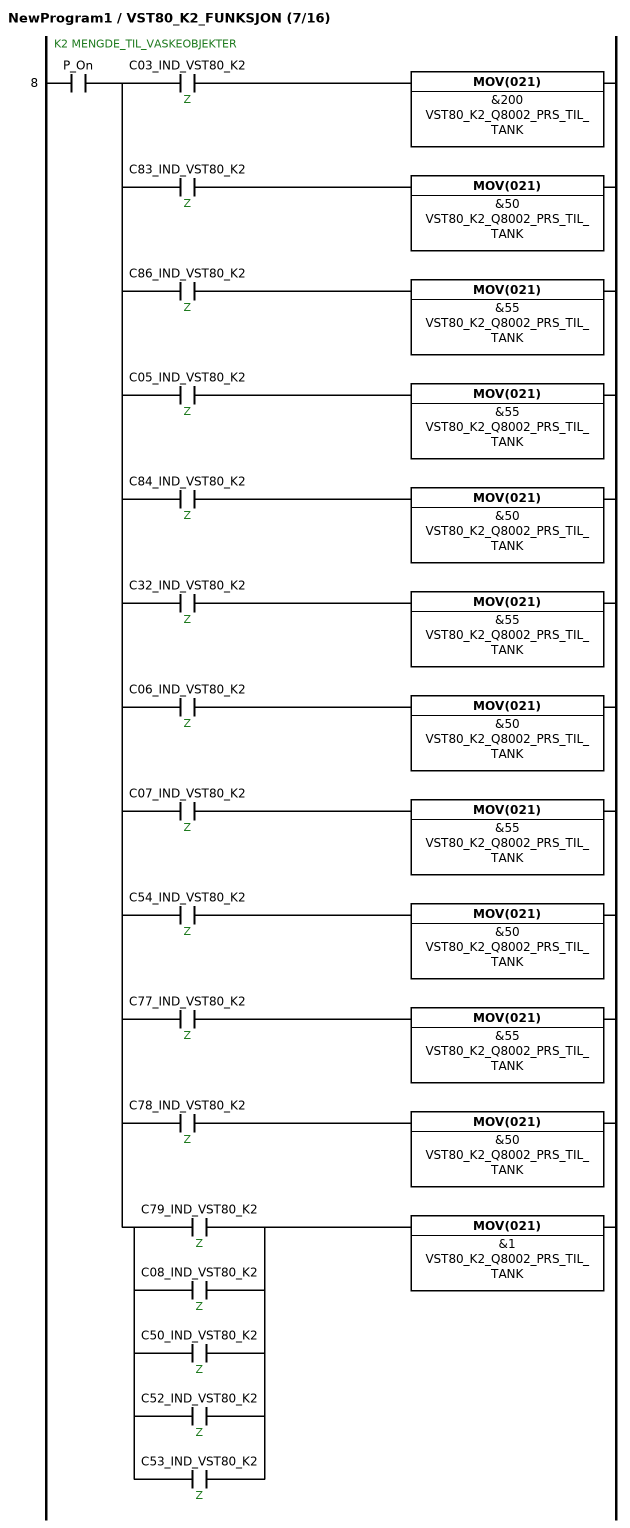
; [picture p240: NewProgram1 / VST80_K2_FUNKSJON, rungs 8-8]
; rung 8: K2 MENGDE_TIL_VASKEOBJEKTER
LD P_On
OUT TR0
AND C03_IND_VST80_K2  ; Z
MOV(021) &200 VST80_K2_Q8002_PRS_TIL_TANK
LD TR0
AND C83_IND_VST80_K2  ; Z
MOV(021) &50 VST80_K2_Q8002_PRS_TIL_TANK
LD TR0
AND C86_IND_VST80_K2  ; Z
MOV(021) &55 VST80_K2_Q8002_PRS_TIL_TANK
LD TR0
AND C05_IND_VST80_K2  ; Z
MOV(021) &55 VST80_K2_Q8002_PRS_TIL_TANK
LD TR0
AND C84_IND_VST80_K2  ; Z
MOV(021) &50 VST80_K2_Q8002_PRS_TIL_TANK
LD TR0
AND C32_IND_VST80_K2  ; Z
MOV(021) &55 VST80_K2_Q8002_PRS_TIL_TANK
LD TR0
AND C06_IND_VST80_K2  ; Z
MOV(021) &50 VST80_K2_Q8002_PRS_TIL_TANK
LD TR0
AND C07_IND_VST80_K2  ; Z
MOV(021) &55 VST80_K2_Q8002_PRS_TIL_TANK
LD TR0
AND C54_IND_VST80_K2  ; Z
MOV(021) &50 VST80_K2_Q8002_PRS_TIL_TANK
LD TR0
AND C77_IND_VST80_K2  ; Z
MOV(021) &55 VST80_K2_Q8002_PRS_TIL_TANK
LD TR0
AND C78_IND_VST80_K2  ; Z
MOV(021) &50 VST80_K2_Q8002_PRS_TIL_TANK
LD TR0
LD C79_IND_VST80_K2  ; Z
OR C08_IND_VST80_K2  ; Z
OR C50_IND_VST80_K2  ; Z
OR C52_IND_VST80_K2  ; Z
OR C53_IND_VST80_K2  ; Z
ANDLD
MOV(021) &1 VST80_K2_Q8002_PRS_TIL_TANK

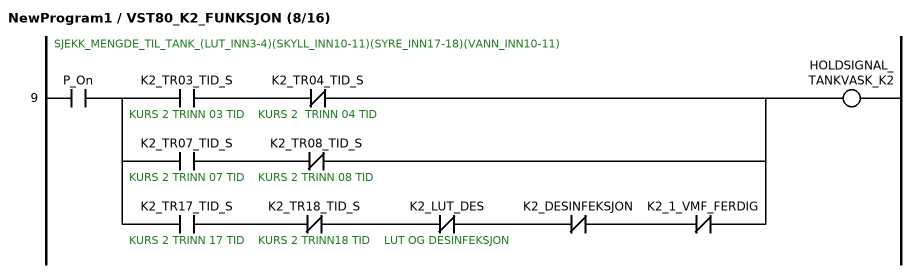
; rung 9: SJEKK_MENGDE_TIL_TANK_(LUT_INN3-4)(SKYLL_INN10-11)(SYRE_INN17-18)(VANN_INN10-11)
LD P_On
LD K2_TR03_TID_S  ; KURS 2 TRINN 03 TID
ANDNOT K2_TR04_TID_S  ; KURS 2  TRINN 04 TID
LD K2_TR07_TID_S  ; KURS 2 TRINN 07 TID
ANDNOT K2_TR08_TID_S  ; KURS 2 TRINN 08 TID
ORLD
LD K2_TR17_TID_S  ; KURS 2 TRINN 17 TID
ANDNOT K2_TR18_TID_S  ; KURS 2 TRINN18 TID
ANDNOT K2_LUT_DES  ; LUT OG DESINFEKSJON
ANDNOT K2_DESINFEKSJON
ANDNOT K2_1_VMF_FERDIG
ORLD
ANDLD
OUT HOLDSIGNAL_TANKVASK_K2

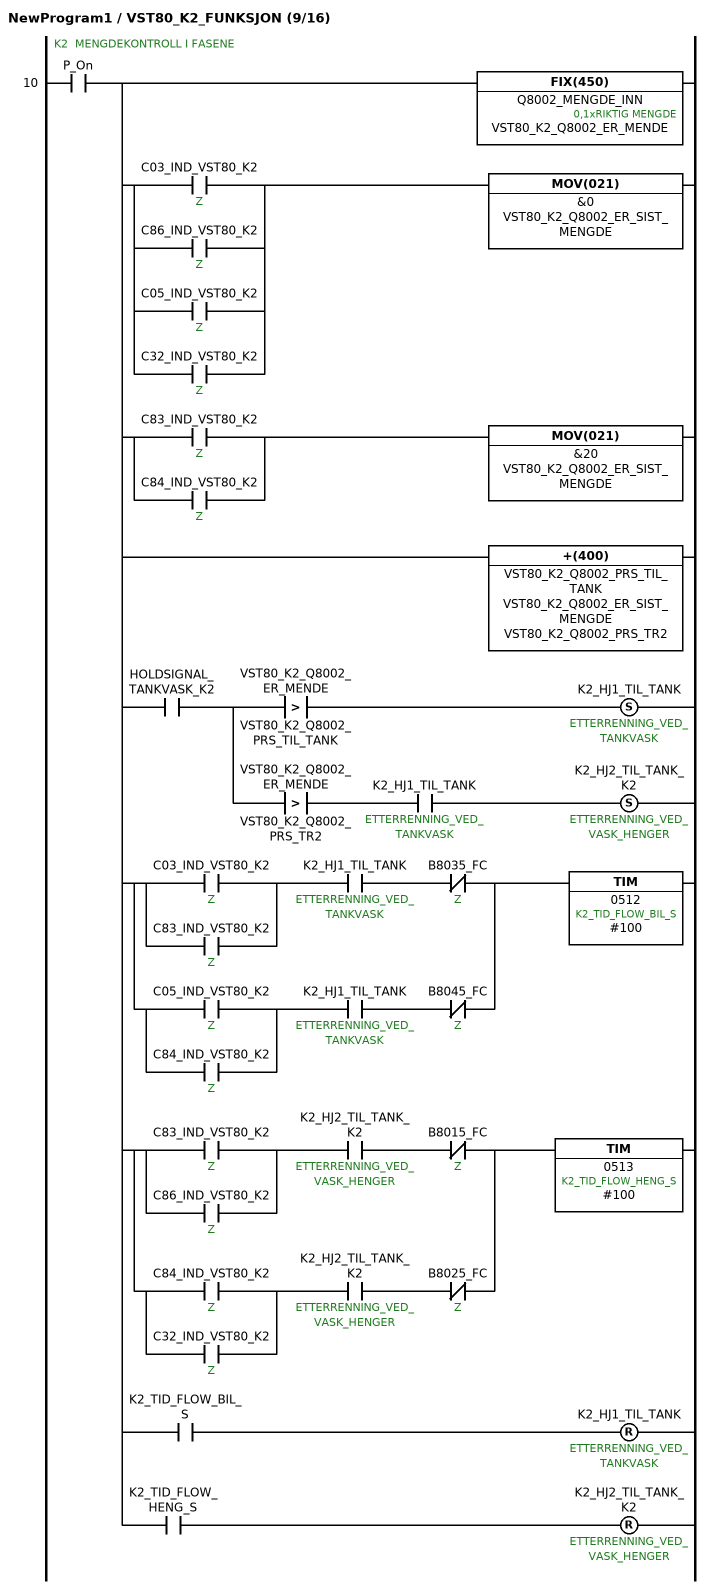
; rung 10: K2  MENGDEKONTROLL I FASENE
LD P_On
OUT TR0
FIX(450) Q8002_MENGDE_INN VST80_K2_Q8002_ER_MENDE  ; 0,1xRIKTIG MENGDE
LD C03_IND_VST80_K2  ; Z
OR C86_IND_VST80_K2  ; Z
OR C05_IND_VST80_K2  ; Z
OR C32_IND_VST80_K2  ; Z
ANDLD
MOV(021) &0 VST80_K2_Q8002_ER_SIST_MENGDE
LD TR0
LD C83_IND_VST80_K2  ; Z
OR C84_IND_VST80_K2  ; Z
ANDLD
MOV(021) &20 VST80_K2_Q8002_ER_SIST_MENGDE
LD TR0
+(400) VST80_K2_Q8002_PRS_TIL_TANK VST80_K2_Q8002_ER_SIST_MENGDE VST80_K2_Q8002_PRS_TR2
AND HOLDSIGNAL_TANKVASK_K2
OUT TR1
AND>(320) VST80_K2_Q8002_ER_MENDE VST80_K2_Q8002_PRS_TIL_TANK
SET K2_HJ1_TIL_TANK  ; ETTERRENNING_VED_TANKVASK
LD TR1
AND>(320) VST80_K2_Q8002_ER_MENDE VST80_K2_Q8002_PRS_TR2
AND K2_HJ1_TIL_TANK  ; ETTERRENNING_VED_TANKVASK
SET K2_HJ2_TIL_TANK_K2  ; ETTERRENNING_VED_VASK_HENGER
LD TR0
LD C03_IND_VST80_K2  ; Z
OR C83_IND_VST80_K2  ; Z
AND K2_HJ1_TIL_TANK  ; ETTERRENNING_VED_TANKVASK
ANDNOT B8035_FC  ; Z
LD C05_IND_VST80_K2  ; Z
OR C84_IND_VST80_K2  ; Z
AND K2_HJ1_TIL_TANK  ; ETTERRENNING_VED_TANKVASK
ANDNOT B8045_FC  ; Z
ORLD
ANDLD
TIM 0512 #100  ; K2_TID_FLOW_BIL_S
LD TR0
LD C83_IND_VST80_K2  ; Z
OR C86_IND_VST80_K2  ; Z
AND K2_HJ2_TIL_TANK_K2  ; ETTERRENNING_VED_VASK_HENGER
ANDNOT B8015_FC  ; Z
LD C84_IND_VST80_K2  ; Z
OR C32_IND_VST80_K2  ; Z
AND K2_HJ2_TIL_TANK_K2  ; ETTERRENNING_VED_VASK_HENGER
ANDNOT B8025_FC  ; Z
ORLD
ANDLD
TIM 0513 #100  ; K2_TID_FLOW_HENG_S
LD TR0
AND K2_TID_FLOW_BIL_S
RSET K2_HJ1_TIL_TANK  ; ETTERRENNING_VED_TANKVASK
LD TR0
AND K2_TID_FLOW_HENG_S
RSET K2_HJ2_TIL_TANK_K2  ; ETTERRENNING_VED_VASK_HENGER

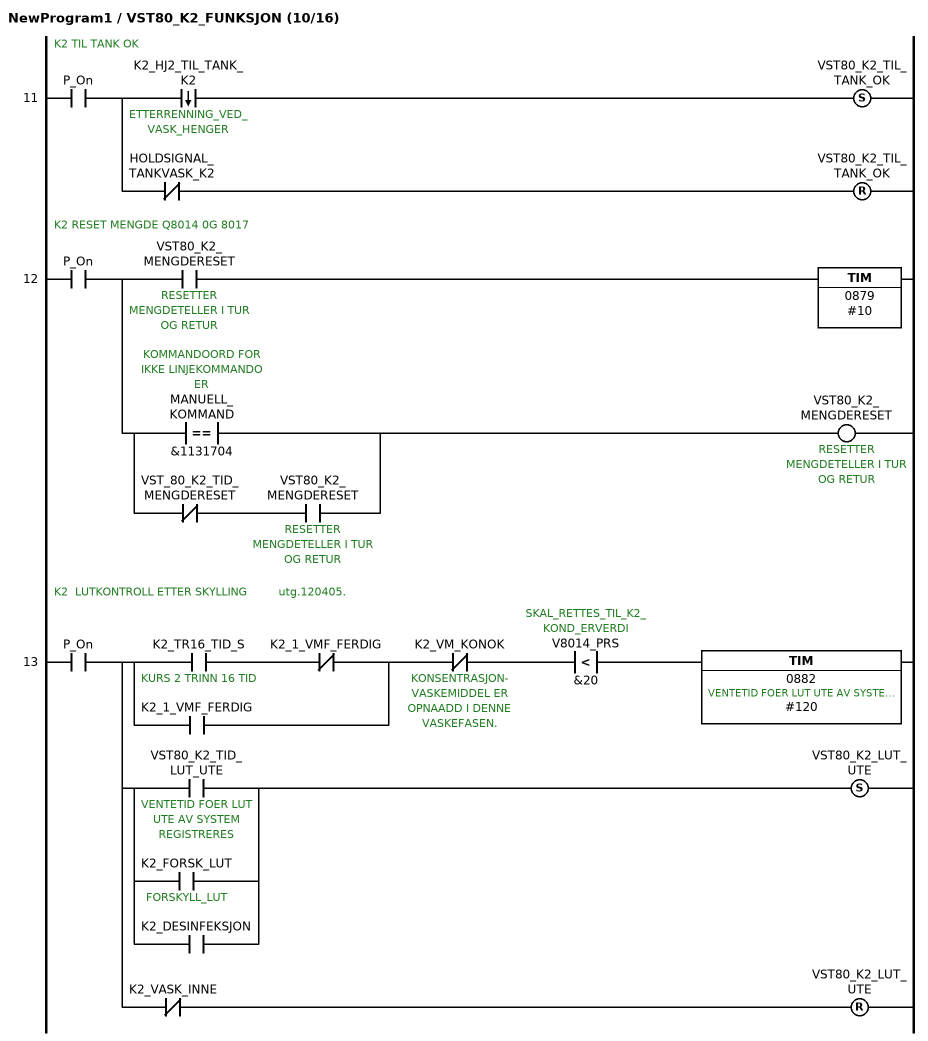
; rung 11: K2 TIL TANK OK
LD P_On
OUT TR0
%AND K2_HJ2_TIL_TANK_K2  ; ETTERRENNING_VED_VASK_HENGER
SET VST80_K2_TIL_TANK_OK
LD TR0
ANDNOT HOLDSIGNAL_TANKVASK_K2
RSET VST80_K2_TIL_TANK_OK
; rung 12: K2 RESET MENGDE Q8014 0G 8017
LD P_On
OUT TR0
AND VST80_K2_MENGDERESET  ; RESETTER MENGDETELLER I TUR OG RETUR
TIM 0879 #10
LD TR0
LD=L(301) MANUELL_KOMMAND &1131704  ; KOMMANDOORD FOR IKKE LINJEKOMMANDOER
LDNOT VST_80_K2_TID_MENGDERESET
AND VST80_K2_MENGDERESET  ; RESETTER MENGDETELLER I TUR OG RETUR
ORLD
ANDLD
OUT VST80_K2_MENGDERESET  ; RESETTER MENGDETELLER I TUR OG RETUR
; rung 13: K2  LUTKONTROLL ETTER SKYLLING         utg.120405.
LD P_On
OUT TR0
LD K2_TR16_TID_S  ; KURS 2 TRINN 16 TID
ANDNOT K2_1_VMF_FERDIG
OR K2_1_VMF_FERDIG
ANDLD
ANDNOT K2_VM_KONOK  ; KONSENTRASJON-VASKEMIDDEL ER OPNAADD I DENNE VASKEFASEN.
AND<(310) V8014_PRS &20  ; SKAL_RETTES_TIL_K2_KOND_ERVERDI
TIM 0882 #120  ; VENTETID FOER LUT UTE AV SYSTEM REGISTRERES
LD TR0
LD VST80_K2_TID_LUT_UTE  ; VENTETID FOER LUT UTE AV SYSTEM REGISTRERES
OR K2_FORSK_LUT  ; FORSKYLL_LUT
OR K2_DESINFEKSJON
ANDLD
SET VST80_K2_LUT_UTE
LD TR0
ANDNOT K2_VASK_INNE
RSET VST80_K2_LUT_UTE

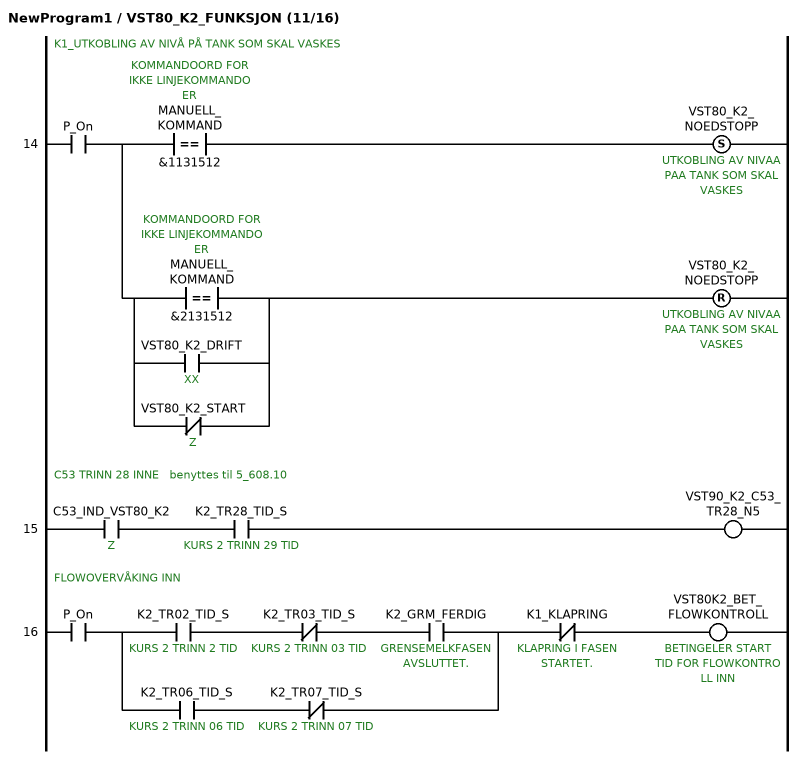
; rung 14: K1_UTKOBLING AV NIVÅ PÅ TANK SOM SKAL VASKES
LD P_On
OUT TR0
AND=L(301) MANUELL_KOMMAND &1131512  ; KOMMANDOORD FOR IKKE LINJEKOMMANDOER
SET VST80_K2_NOEDSTOPP  ; UTKOBLING AV NIVAA PAA TANK SOM SKAL VASKES
LD TR0
LD=L(301) MANUELL_KOMMAND &2131512  ; KOMMANDOORD FOR IKKE LINJEKOMMANDOER
OR VST80_K2_DRIFT  ; XX
ORNOT VST80_K2_START  ; Z
ANDLD
RSET VST80_K2_NOEDSTOPP  ; UTKOBLING AV NIVAA PAA TANK SOM SKAL VASKES
; rung 15: C53 TRINN 28 INNE   benyttes til 5_608.10
LD C53_IND_VST80_K2  ; Z
AND K2_TR28_TID_S  ; KURS 2 TRINN 29 TID
OUT VST90_K2_C53_TR28_N5
; rung 16: FLOWOVERVÅKING INN
LD P_On
LD K2_TR02_TID_S  ; KURS 2 TRINN 2 TID
ANDNOT K2_TR03_TID_S  ; KURS 2 TRINN 03 TID
AND K2_GRM_FERDIG  ; GRENSEMELKFASEN AVSLUTTET.
LD K2_TR06_TID_S  ; KURS 2 TRINN 06 TID
ANDNOT K2_TR07_TID_S  ; KURS 2 TRINN 07 TID
ORLD
ANDLD
ANDNOT K1_KLAPRING  ; KLAPRING I FASEN STARTET.
OUT VST80K2_BET_FLOWKONTROLL  ; BETINGELER START TID FOR FLOWKONTROLL INN

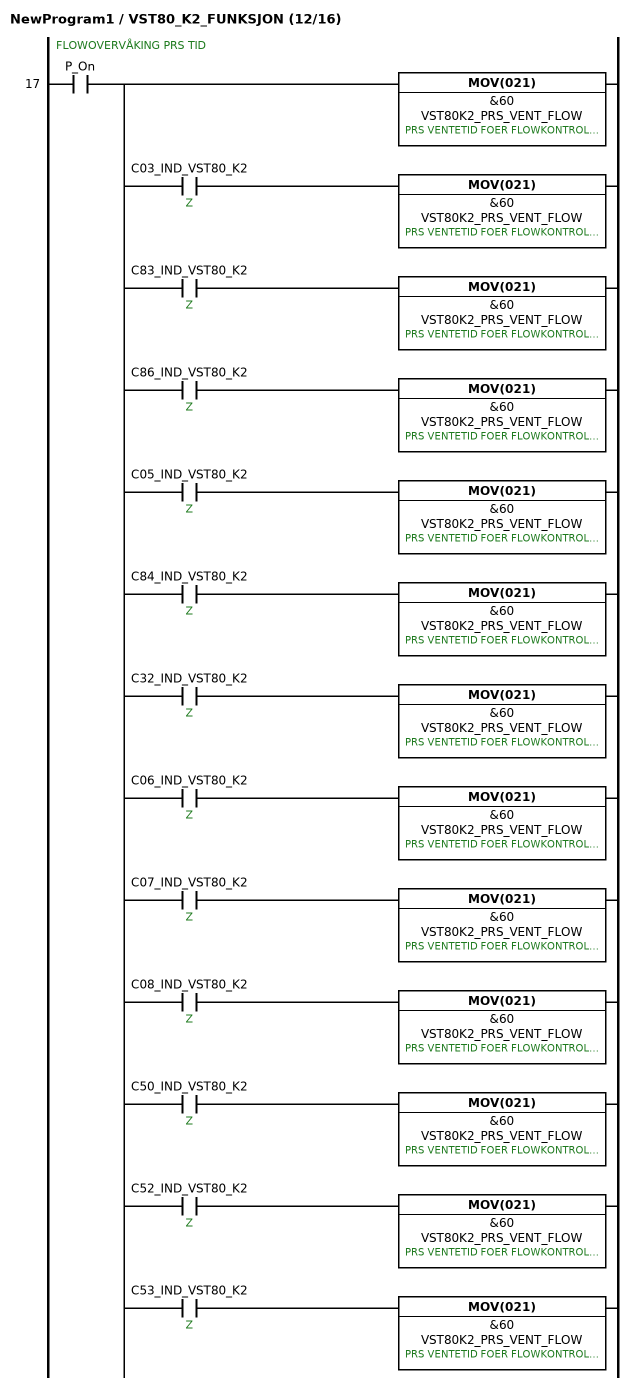

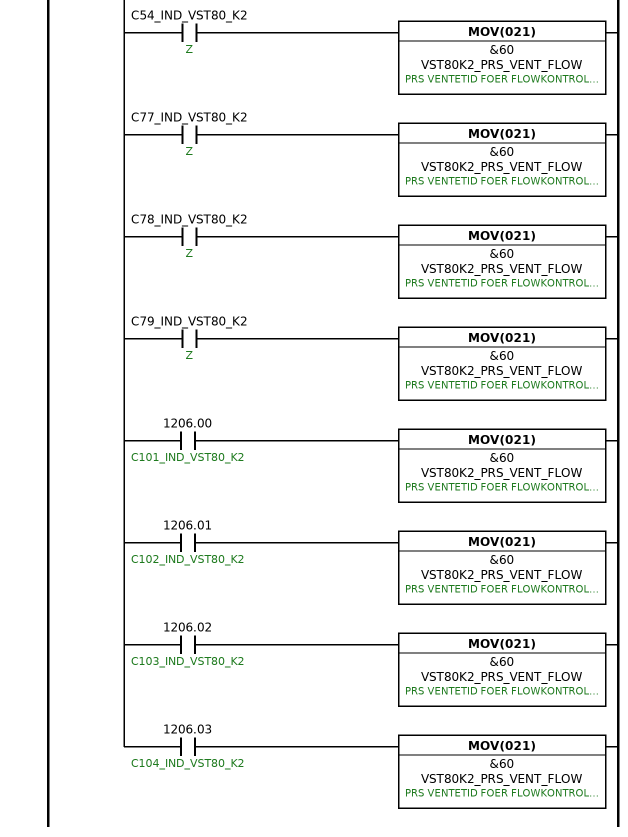
; rung 17: FLOWOVERVÅKING PRS TID
LD P_On
OUT TR0
MOV(021) &60 VST80K2_PRS_VENT_FLOW  ; PRS VENTETID FOER FLOWKONTROLL STARTER
AND C03_IND_VST80_K2  ; Z
MOV(021) &60 VST80K2_PRS_VENT_FLOW  ; PRS VENTETID FOER FLOWKONTROLL STARTER
LD TR0
AND C83_IND_VST80_K2  ; Z
MOV(021) &60 VST80K2_PRS_VENT_FLOW  ; PRS VENTETID FOER FLOWKONTROLL STARTER
LD TR0
AND C86_IND_VST80_K2  ; Z
MOV(021) &60 VST80K2_PRS_VENT_FLOW  ; PRS VENTETID FOER FLOWKONTROLL STARTER
LD TR0
AND C05_IND_VST80_K2  ; Z
MOV(021) &60 VST80K2_PRS_VENT_FLOW  ; PRS VENTETID FOER FLOWKONTROLL STARTER
LD TR0
AND C84_IND_VST80_K2  ; Z
MOV(021) &60 VST80K2_PRS_VENT_FLOW  ; PRS VENTETID FOER FLOWKONTROLL STARTER
LD TR0
AND C32_IND_VST80_K2  ; Z
MOV(021) &60 VST80K2_PRS_VENT_FLOW  ; PRS VENTETID FOER FLOWKONTROLL STARTER
LD TR0
AND C06_IND_VST80_K2  ; Z
MOV(021) &60 VST80K2_PRS_VENT_FLOW  ; PRS VENTETID FOER FLOWKONTROLL STARTER
LD TR0
AND C07_IND_VST80_K2  ; Z
MOV(021) &60 VST80K2_PRS_VENT_FLOW  ; PRS VENTETID FOER FLOWKONTROLL STARTER
LD TR0
AND C08_IND_VST80_K2  ; Z
MOV(021) &60 VST80K2_PRS_VENT_FLOW  ; PRS VENTETID FOER FLOWKONTROLL STARTER
LD TR0
AND C50_IND_VST80_K2  ; Z
MOV(021) &60 VST80K2_PRS_VENT_FLOW  ; PRS VENTETID FOER FLOWKONTROLL STARTER
LD TR0
AND C52_IND_VST80_K2  ; Z
MOV(021) &60 VST80K2_PRS_VENT_FLOW  ; PRS VENTETID FOER FLOWKONTROLL STARTER
LD TR0
AND C53_IND_VST80_K2  ; Z
MOV(021) &60 VST80K2_PRS_VENT_FLOW  ; PRS VENTETID FOER FLOWKONTROLL STARTER
LD TR0
AND C54_IND_VST80_K2  ; Z
MOV(021) &60 VST80K2_PRS_VENT_FLOW  ; PRS VENTETID FOER FLOWKONTROLL STARTER
LD TR0
AND C77_IND_VST80_K2  ; Z
MOV(021) &60 VST80K2_PRS_VENT_FLOW  ; PRS VENTETID FOER FLOWKONTROLL STARTER
LD TR0
AND C78_IND_VST80_K2  ; Z
MOV(021) &60 VST80K2_PRS_VENT_FLOW  ; PRS VENTETID FOER FLOWKONTROLL STARTER
LD TR0
AND C79_IND_VST80_K2  ; Z
MOV(021) &60 VST80K2_PRS_VENT_FLOW  ; PRS VENTETID FOER FLOWKONTROLL STARTER
LD TR0
AND 1206.00  ; C101_IND_VST80_K2
MOV(021) &60 VST80K2_PRS_VENT_FLOW  ; PRS VENTETID FOER FLOWKONTROLL STARTER
LD TR0
AND 1206.01  ; C102_IND_VST80_K2
MOV(021) &60 VST80K2_PRS_VENT_FLOW  ; PRS VENTETID FOER FLOWKONTROLL STARTER
LD TR0
AND 1206.02  ; C103_IND_VST80_K2
MOV(021) &60 VST80K2_PRS_VENT_FLOW  ; PRS VENTETID FOER FLOWKONTROLL STARTER
LD TR0
AND 1206.03  ; C104_IND_VST80_K2
MOV(021) &60 VST80K2_PRS_VENT_FLOW  ; PRS VENTETID FOER FLOWKONTROLL STARTER

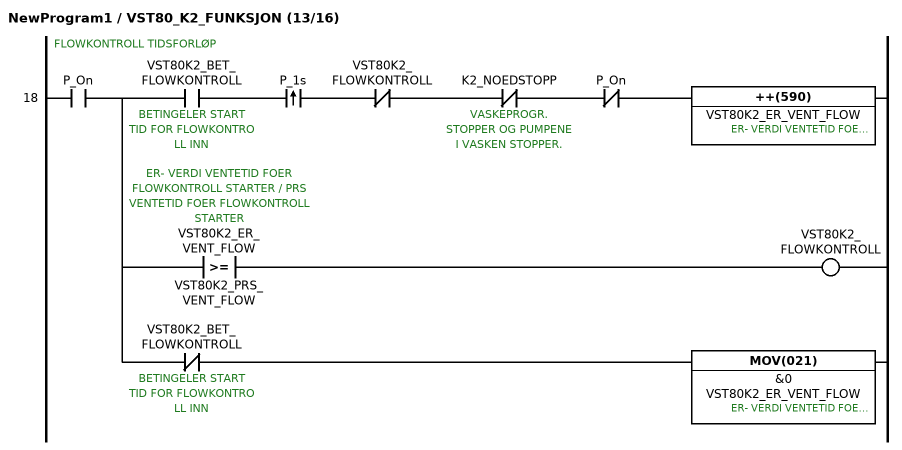
; rung 18: FLOWKONTROLL TIDSFORLØP
LD P_On
OUT TR0
AND VST80K2_BET_FLOWKONTROLL  ; BETINGELER START TID FOR FLOWKONTROLL INN
@AND P_1s
ANDNOT VST80K2_FLOWKONTROLL
ANDNOT K2_NOEDSTOPP  ; VASKEPROGR. STOPPER OG PUMPENE I VASKEN STOPPER.
ANDNOT P_On
++(590) VST80K2_ER_VENT_FLOW  ; ER- VERDI VENTETID FOER FLOWKONTROLL STARTER
LD TR0
AND>=(325) VST80K2_ER_VENT_FLOW VST80K2_PRS_VENT_FLOW  ; ER- VERDI VENTETID FOER FLOWKONTROLL STARTER, PRS VENTETID FOER FLOWKONTROLL STARTER
OUT VST80K2_FLOWKONTROLL
LD TR0
ANDNOT VST80K2_BET_FLOWKONTROLL  ; BETINGELER START TID FOR FLOWKONTROLL INN
MOV(021) &0 VST80K2_ER_VENT_FLOW  ; ER- VERDI VENTETID FOER FLOWKONTROLL STARTER

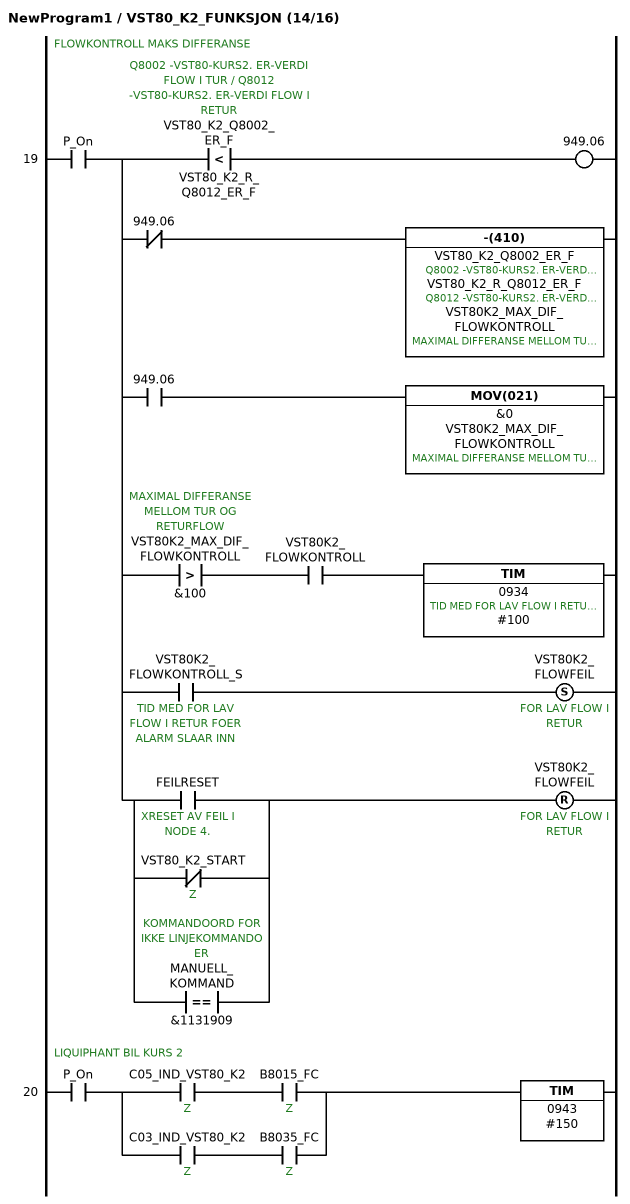
; rung 19: FLOWKONTROLL MAKS DIFFERANSE
LD P_On
OUT TR0
AND<(310) VST80_K2_Q8002_ER_F VST80_K2_R_Q8012_ER_F  ; Q8002 -VST80-KURS2. ER-VERDI FLOW I TUR, Q8012 -VST80-KURS2. ER-VERDI FLOW I RETUR
OUT 949.06
LD TR0
ANDNOT 949.06
-(410) VST80_K2_Q8002_ER_F VST80_K2_R_Q8012_ER_F VST80K2_MAX_DIF_FLOWKONTROLL  ; Q8002 -VST80-KURS2. ER-VERDI FLOW I TUR, Q8012 -VST80-KURS2. ER-VERDI FLOW I RETUR, MAXIMAL DIFFERANSE MELLOM TUR OG RETURFLOW
LD TR0
AND 949.06
MOV(021) &0 VST80K2_MAX_DIF_FLOWKONTROLL  ; MAXIMAL DIFFERANSE MELLOM TUR OG RETURFLOW
LD TR0
AND>(320) VST80K2_MAX_DIF_FLOWKONTROLL &100  ; MAXIMAL DIFFERANSE MELLOM TUR OG RETURFLOW
AND VST80K2_FLOWKONTROLL
TIM 0934 #100  ; TID MED FOR LAV FLOW I RETUR FOER ALARM SLAAR INN
LD TR0
AND VST80K2_FLOWKONTROLL_S  ; TID MED FOR LAV FLOW I RETUR FOER ALARM SLAAR INN
SET VST80K2_FLOWFEIL  ; FOR LAV FLOW I RETUR
LD TR0
LD FEILRESET  ; XRESET AV FEIL I NODE 4.
ORNOT VST80_K2_START  ; Z
OR=L(301) MANUELL_KOMMAND &1131909  ; KOMMANDOORD FOR IKKE LINJEKOMMANDOER
ANDLD
RSET VST80K2_FLOWFEIL  ; FOR LAV FLOW I RETUR
; rung 20: LIQUIPHANT BIL KURS 2
LD P_On
LD C05_IND_VST80_K2  ; Z
AND B8015_FC  ; Z
LD C03_IND_VST80_K2  ; Z
AND B8035_FC  ; Z
ORLD
ANDLD
TIM 0943 #150

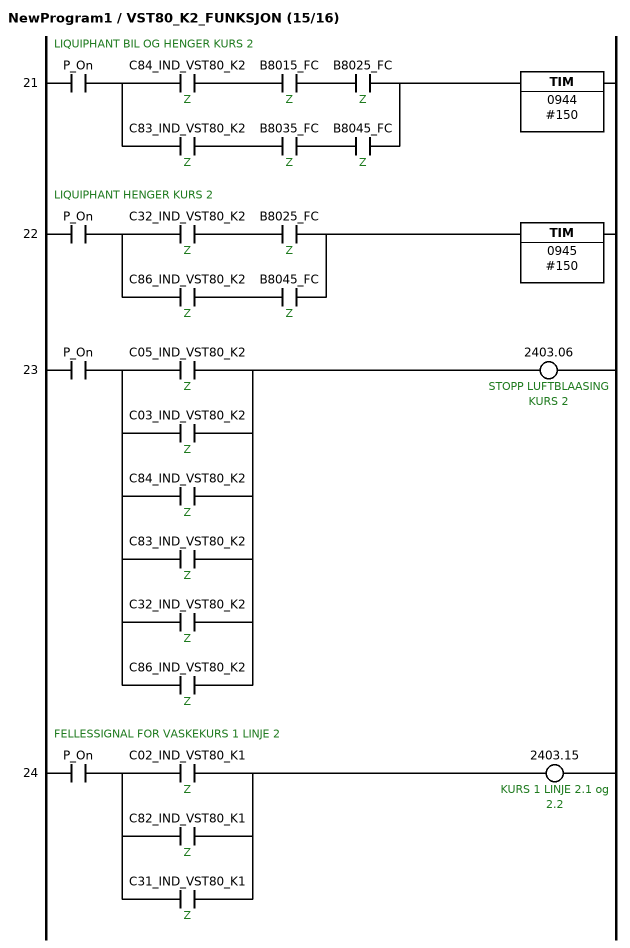
; rung 21: LIQUIPHANT BIL OG HENGER KURS 2
LD P_On
LD C84_IND_VST80_K2  ; Z
AND B8015_FC  ; Z
AND B8025_FC  ; Z
LD C83_IND_VST80_K2  ; Z
AND B8035_FC  ; Z
AND B8045_FC  ; Z
ORLD
ANDLD
TIM 0944 #150
; rung 22: LIQUIPHANT HENGER KURS 2
LD P_On
LD C32_IND_VST80_K2  ; Z
AND B8025_FC  ; Z
LD C86_IND_VST80_K2  ; Z
AND B8045_FC  ; Z
ORLD
ANDLD
TIM 0945 #150
; rung 23
LD P_On
LD C05_IND_VST80_K2  ; Z
OR C03_IND_VST80_K2  ; Z
OR C84_IND_VST80_K2  ; Z
OR C83_IND_VST80_K2  ; Z
OR C32_IND_VST80_K2  ; Z
OR C86_IND_VST80_K2  ; Z
ANDLD
OUT 2403.06  ; STOPP LUFTBLAASING KURS 2
; rung 24: FELLESSIGNAL FOR VASKEKURS 1 LINJE 2
LD P_On
LD C02_IND_VST80_K1  ; Z
OR C82_IND_VST80_K1  ; Z
OR C31_IND_VST80_K1  ; Z
ANDLD
OUT 2403.15  ; KURS 1 LINJE 2.1 og 2.2

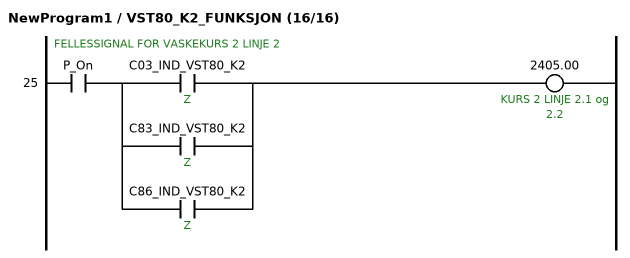
; rung 25: FELLESSIGNAL FOR VASKEKURS 2 LINJE 2
LD P_On
LD C03_IND_VST80_K2  ; Z
OR C83_IND_VST80_K2  ; Z
OR C86_IND_VST80_K2  ; Z
ANDLD
OUT 2405.00  ; KURS 2 LINJE 2.1 og 2.2

### Section VST80_K2_OBJEKTER
; Styring av objektene i kurs K1

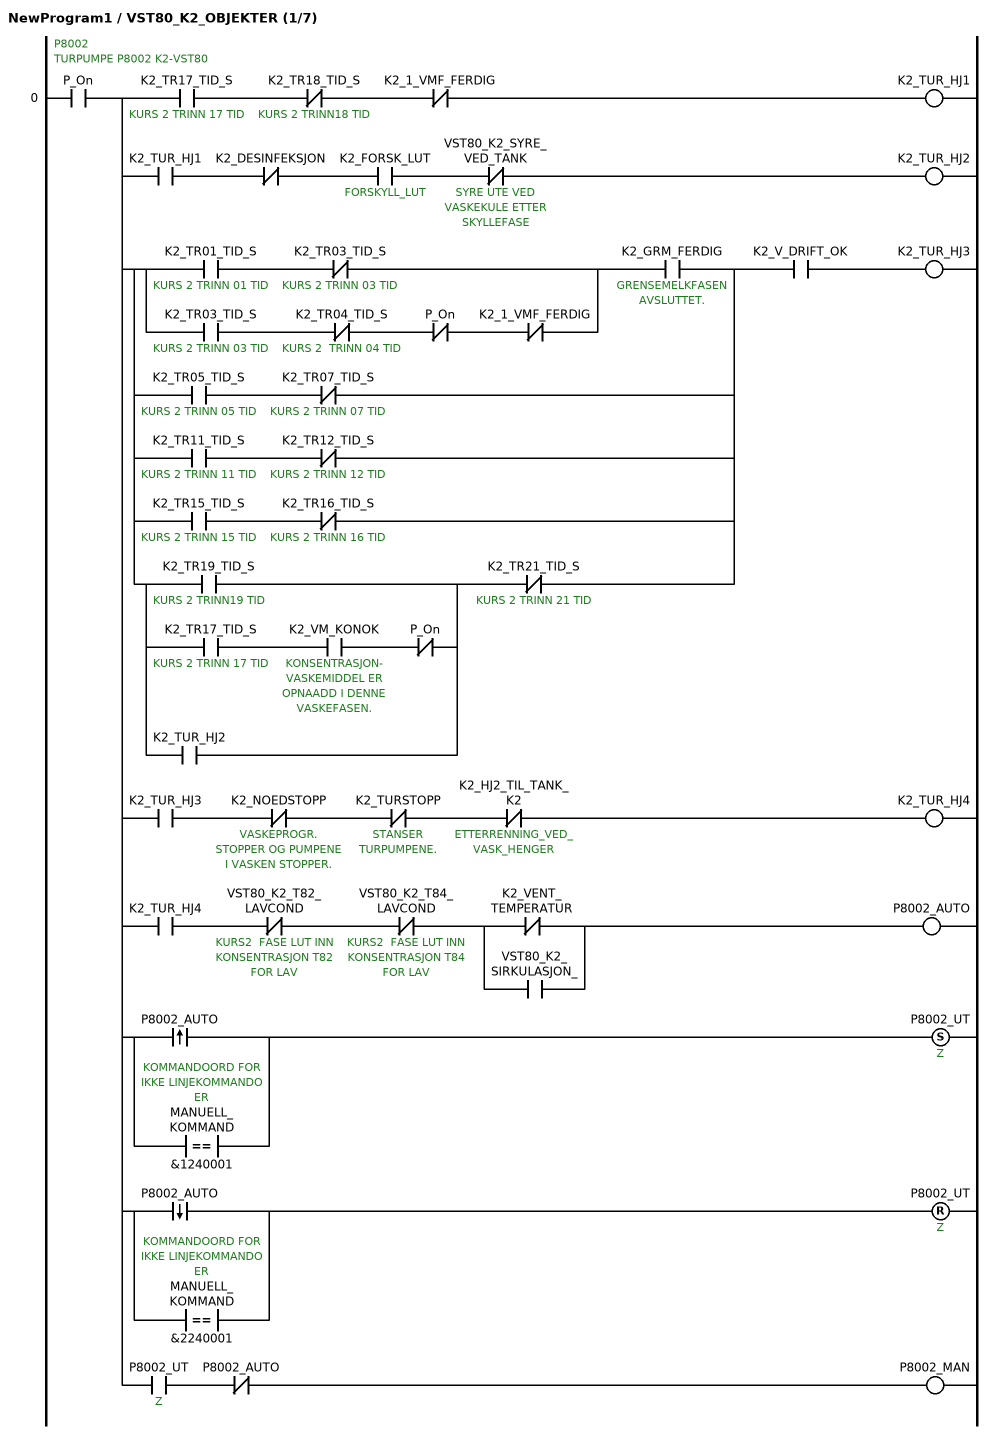
; rung 0: P8002 / TURPUMPE P8002 K2-VST80
LD P_On
OUT TR0
AND K2_TR17_TID_S  ; KURS 2 TRINN 17 TID
ANDNOT K2_TR18_TID_S  ; KURS 2 TRINN18 TID
ANDNOT K2_1_VMF_FERDIG
OUT K2_TUR_HJ1
LD TR0
AND K2_TUR_HJ1
ANDNOT K2_DESINFEKSJON
AND K2_FORSK_LUT  ; FORSKYLL_LUT
ANDNOT VST80_K2_SYRE_VED_TANK  ; SYRE UTE VED VASKEKULE ETTER SKYLLEFASE
OUT K2_TUR_HJ2
LD TR0
LD K2_TR01_TID_S  ; KURS 2 TRINN 01 TID
ANDNOT K2_TR03_TID_S  ; KURS 2 TRINN 03 TID
LD K2_TR03_TID_S  ; KURS 2 TRINN 03 TID
ANDNOT K2_TR04_TID_S  ; KURS 2  TRINN 04 TID
ANDNOT P_On
ANDNOT K2_1_VMF_FERDIG
ORLD
AND K2_GRM_FERDIG  ; GRENSEMELKFASEN AVSLUTTET.
LD K2_TR05_TID_S  ; KURS 2 TRINN 05 TID
ANDNOT K2_TR07_TID_S  ; KURS 2 TRINN 07 TID
ORLD
LD K2_TR11_TID_S  ; KURS 2 TRINN 11 TID
ANDNOT K2_TR12_TID_S  ; KURS 2 TRINN 12 TID
ORLD
LD K2_TR15_TID_S  ; KURS 2 TRINN 15 TID
ANDNOT K2_TR16_TID_S  ; KURS 2 TRINN 16 TID
ORLD
LD K2_TR19_TID_S  ; KURS 2 TRINN19 TID
LD K2_TR17_TID_S  ; KURS 2 TRINN 17 TID
AND K2_VM_KONOK  ; KONSENTRASJON-VASKEMIDDEL ER OPNAADD I DENNE VASKEFASEN.
ANDNOT P_On
ORLD
OR K2_TUR_HJ2
ANDNOT K2_TR21_TID_S  ; KURS 2 TRINN 21 TID
ORLD
ANDLD
AND K2_V_DRIFT_OK
OUT K2_TUR_HJ3
LD TR0
AND K2_TUR_HJ3
ANDNOT K2_NOEDSTOPP  ; VASKEPROGR. STOPPER OG PUMPENE I VASKEN STOPPER.
ANDNOT K2_TURSTOPP  ; STANSER TURPUMPENE.
ANDNOT K2_HJ2_TIL_TANK_K2  ; ETTERRENNING_VED_VASK_HENGER
OUT K2_TUR_HJ4
LD TR0
AND K2_TUR_HJ4
ANDNOT VST80_K2_T82_LAVCOND  ; KURS2  FASE LUT INN KONSENTRASJON T82 FOR LAV
ANDNOT VST80_K2_T84_LAVCOND  ; KURS2  FASE LUT INN KONSENTRASJON T84 FOR LAV
LDNOT K2_VENT_TEMPERATUR
OR VST80_K2_SIRKULASJON_
ANDLD
OUT P8002_AUTO
LD TR0
@LD P8002_AUTO
OR=L(301) MANUELL_KOMMAND &1240001  ; KOMMANDOORD FOR IKKE LINJEKOMMANDOER
ANDLD
SET P8002_UT  ; Z
LD TR0
%LD P8002_AUTO
OR=L(301) MANUELL_KOMMAND &2240001  ; KOMMANDOORD FOR IKKE LINJEKOMMANDOER
ANDLD
RSET P8002_UT  ; Z
LD TR0
AND P8002_UT  ; Z
ANDNOT P8002_AUTO
OUT P8002_MAN

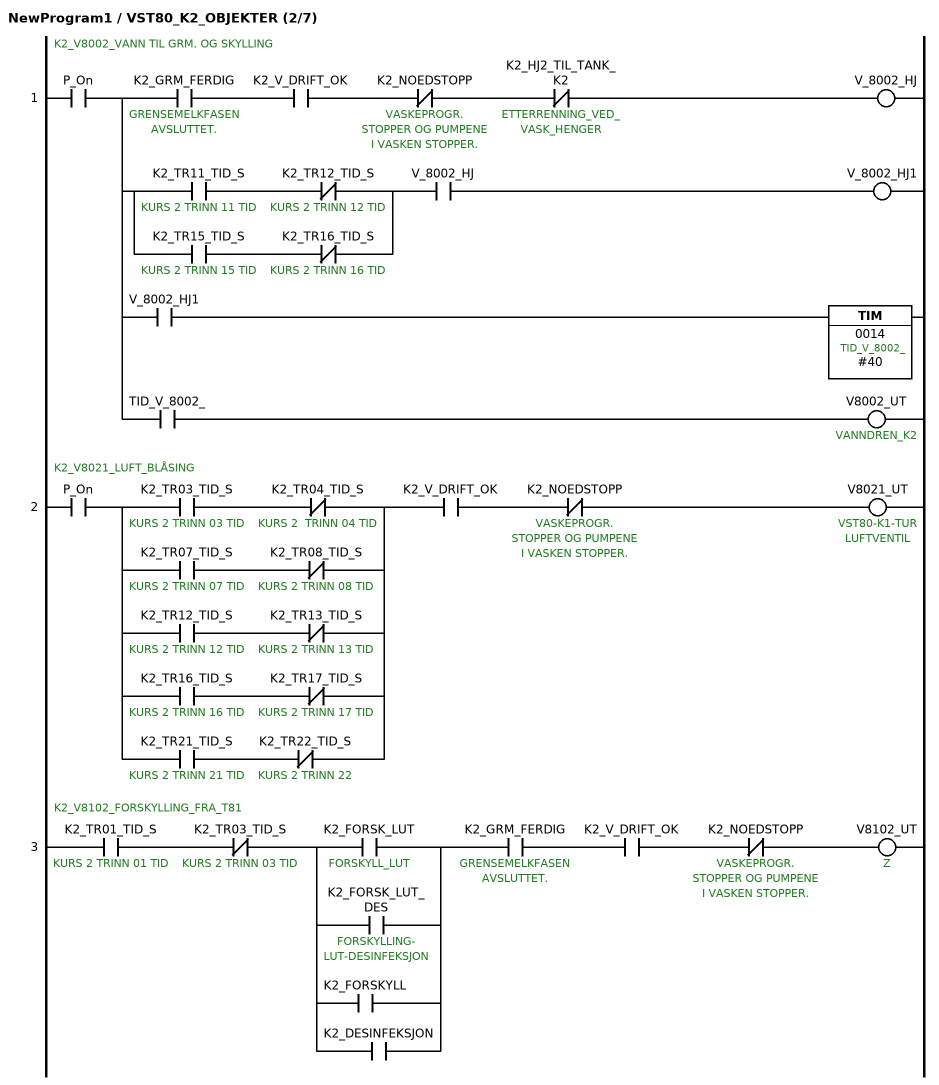
; rung 1: K2_V8002_VANN TIL GRM. OG SKYLLING
LD P_On
OUT TR0
AND K2_GRM_FERDIG  ; GRENSEMELKFASEN AVSLUTTET.
AND K2_V_DRIFT_OK
ANDNOT K2_NOEDSTOPP  ; VASKEPROGR. STOPPER OG PUMPENE I VASKEN STOPPER.
ANDNOT K2_HJ2_TIL_TANK_K2  ; ETTERRENNING_VED_VASK_HENGER
OUT V_8002_HJ
LD TR0
LD K2_TR11_TID_S  ; KURS 2 TRINN 11 TID
ANDNOT K2_TR12_TID_S  ; KURS 2 TRINN 12 TID
LD K2_TR15_TID_S  ; KURS 2 TRINN 15 TID
ANDNOT K2_TR16_TID_S  ; KURS 2 TRINN 16 TID
ORLD
ANDLD
AND V_8002_HJ
OUT V_8002_HJ1
LD TR0
AND V_8002_HJ1
TIM 0014 #40  ; TID_V_8002_
LD TR0
AND TID_V_8002_
OUT V8002_UT  ; VANNDREN_K2
; rung 2: K2_V8021_LUFT_BLÅSING
LD P_On
LD K2_TR03_TID_S  ; KURS 2 TRINN 03 TID
ANDNOT K2_TR04_TID_S  ; KURS 2  TRINN 04 TID
LD K2_TR07_TID_S  ; KURS 2 TRINN 07 TID
ANDNOT K2_TR08_TID_S  ; KURS 2 TRINN 08 TID
ORLD
LD K2_TR12_TID_S  ; KURS 2 TRINN 12 TID
ANDNOT K2_TR13_TID_S  ; KURS 2 TRINN 13 TID
ORLD
LD K2_TR16_TID_S  ; KURS 2 TRINN 16 TID
ANDNOT K2_TR17_TID_S  ; KURS 2 TRINN 17 TID
ORLD
LD K2_TR21_TID_S  ; KURS 2 TRINN 21 TID
ANDNOT K2_TR22_TID_S  ; KURS 2 TRINN 22
ORLD
ANDLD
AND K2_V_DRIFT_OK
ANDNOT K2_NOEDSTOPP  ; VASKEPROGR. STOPPER OG PUMPENE I VASKEN STOPPER.
OUT V8021_UT  ; VST80-K1-TUR LUFTVENTIL
; rung 3: K2_V8102_FORSKYLLING_FRA_T81
LD K2_TR01_TID_S  ; KURS 2 TRINN 01 TID
ANDNOT K2_TR03_TID_S  ; KURS 2 TRINN 03 TID
LD K2_FORSK_LUT  ; FORSKYLL_LUT
OR K2_FORSK_LUT_DES  ; FORSKYLLING- LUT-DESINFEKSJON
OR K2_FORSKYLL
OR K2_DESINFEKSJON
ANDLD
AND K2_GRM_FERDIG  ; GRENSEMELKFASEN AVSLUTTET.
AND K2_V_DRIFT_OK
ANDNOT K2_NOEDSTOPP  ; VASKEPROGR. STOPPER OG PUMPENE I VASKEN STOPPER.
OUT V8102_UT  ; Z

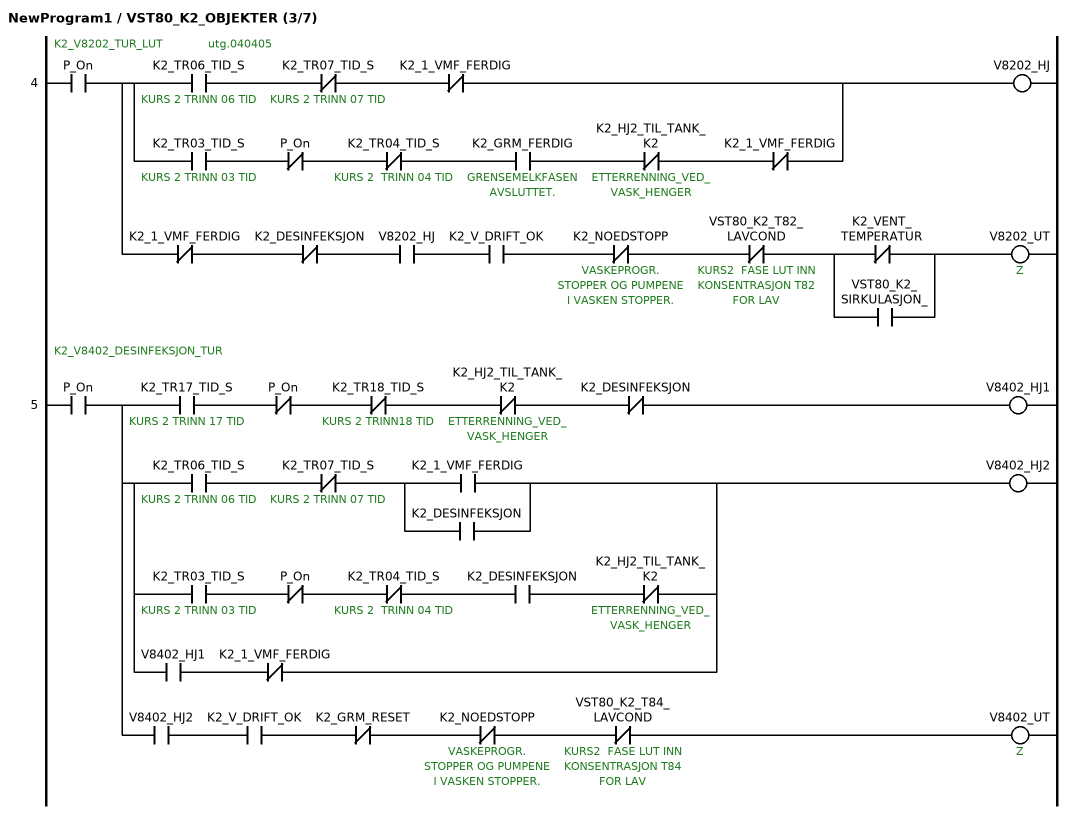
; rung 4: K2_V8202_TUR_LUT             utg.040405
LD P_On
OUT TR0
LD K2_TR06_TID_S  ; KURS 2 TRINN 06 TID
ANDNOT K2_TR07_TID_S  ; KURS 2 TRINN 07 TID
ANDNOT K2_1_VMF_FERDIG
LD K2_TR03_TID_S  ; KURS 2 TRINN 03 TID
ANDNOT P_On
ANDNOT K2_TR04_TID_S  ; KURS 2  TRINN 04 TID
AND K2_GRM_FERDIG  ; GRENSEMELKFASEN AVSLUTTET.
ANDNOT K2_HJ2_TIL_TANK_K2  ; ETTERRENNING_VED_VASK_HENGER
ANDNOT K2_1_VMF_FERDIG
ORLD
ANDLD
OUT V8202_HJ
LD TR0
ANDNOT K2_1_VMF_FERDIG
ANDNOT K2_DESINFEKSJON
AND V8202_HJ
AND K2_V_DRIFT_OK
ANDNOT K2_NOEDSTOPP  ; VASKEPROGR. STOPPER OG PUMPENE I VASKEN STOPPER.
ANDNOT VST80_K2_T82_LAVCOND  ; KURS2  FASE LUT INN KONSENTRASJON T82 FOR LAV
LDNOT K2_VENT_TEMPERATUR
OR VST80_K2_SIRKULASJON_
ANDLD
OUT V8202_UT  ; Z
; rung 5: K2_V8402_DESINFEKSJON_TUR
LD P_On
OUT TR0
AND K2_TR17_TID_S  ; KURS 2 TRINN 17 TID
ANDNOT P_On
ANDNOT K2_TR18_TID_S  ; KURS 2 TRINN18 TID
ANDNOT K2_HJ2_TIL_TANK_K2  ; ETTERRENNING_VED_VASK_HENGER
ANDNOT K2_DESINFEKSJON
OUT V8402_HJ1
LD TR0
LD K2_TR06_TID_S  ; KURS 2 TRINN 06 TID
ANDNOT K2_TR07_TID_S  ; KURS 2 TRINN 07 TID
LD K2_1_VMF_FERDIG
OR K2_DESINFEKSJON
ANDLD
LD K2_TR03_TID_S  ; KURS 2 TRINN 03 TID
ANDNOT P_On
ANDNOT K2_TR04_TID_S  ; KURS 2  TRINN 04 TID
AND K2_DESINFEKSJON
ANDNOT K2_HJ2_TIL_TANK_K2  ; ETTERRENNING_VED_VASK_HENGER
ORLD
LD V8402_HJ1
ANDNOT K2_1_VMF_FERDIG
ORLD
ANDLD
OUT V8402_HJ2
LD TR0
AND V8402_HJ2
AND K2_V_DRIFT_OK
ANDNOT K2_GRM_RESET
ANDNOT K2_NOEDSTOPP  ; VASKEPROGR. STOPPER OG PUMPENE I VASKEN STOPPER.
ANDNOT VST80_K2_T84_LAVCOND  ; KURS2  FASE LUT INN KONSENTRASJON T84 FOR LAV
OUT V8402_UT  ; Z

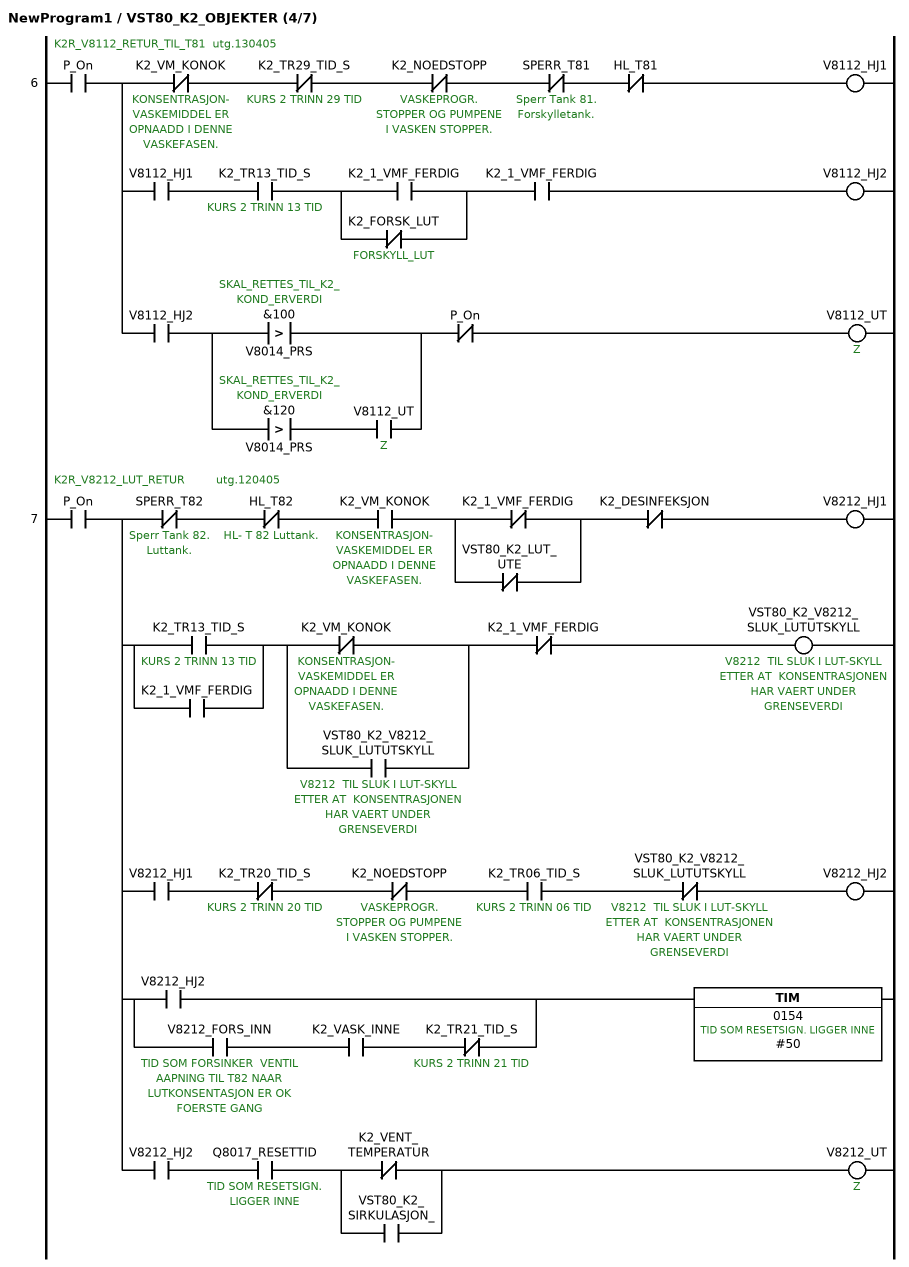
; rung 6: K2R_V8112_RETUR_TIL_T81  utg.130405
LD P_On
OUT TR0
ANDNOT K2_VM_KONOK  ; KONSENTRASJON-VASKEMIDDEL ER OPNAADD I DENNE VASKEFASEN.
ANDNOT K2_TR29_TID_S  ; KURS 2 TRINN 29 TID
ANDNOT K2_NOEDSTOPP  ; VASKEPROGR. STOPPER OG PUMPENE I VASKEN STOPPER.
ANDNOT SPERR_T81  ; Sperr Tank 81. Forskylletank.
ANDNOT HL_T81
OUT V8112_HJ1
LD TR0
AND V8112_HJ1
AND K2_TR13_TID_S  ; KURS 2 TRINN 13 TID
LD K2_1_VMF_FERDIG
ORNOT K2_FORSK_LUT  ; FORSKYLL_LUT
ANDLD
AND K2_1_VMF_FERDIG
OUT V8112_HJ2
LD TR0
AND V8112_HJ2
LD>(320) &100 V8014_PRS  ; SKAL_RETTES_TIL_K2_KOND_ERVERDI
LD>(320) &120 V8014_PRS  ; SKAL_RETTES_TIL_K2_KOND_ERVERDI
AND V8112_UT  ; Z
ORLD
ANDLD
ANDNOT P_On
OUT V8112_UT  ; Z
; rung 7: K2R_V8212_LUT_RETUR         utg.120405
LD P_On
OUT TR0
ANDNOT SPERR_T82  ; Sperr Tank 82. Luttank.
ANDNOT HL_T82  ; HL- T 82 Luttank.
AND K2_VM_KONOK  ; KONSENTRASJON-VASKEMIDDEL ER OPNAADD I DENNE VASKEFASEN.
LDNOT K2_1_VMF_FERDIG
ORNOT VST80_K2_LUT_UTE
ANDLD
ANDNOT K2_DESINFEKSJON
OUT V8212_HJ1
LD TR0
LD K2_TR13_TID_S  ; KURS 2 TRINN 13 TID
OR K2_1_VMF_FERDIG
ANDLD
LDNOT K2_VM_KONOK  ; KONSENTRASJON-VASKEMIDDEL ER OPNAADD I DENNE VASKEFASEN.
OR VST80_K2_V8212_SLUK_LUTUTSKYLL  ; V8212  TIL SLUK I LUT-SKYLL ETTER AT  KONSENTRASJONEN HAR VAERT UNDER  GRENSEVERDI
ANDLD
ANDNOT K2_1_VMF_FERDIG
OUT VST80_K2_V8212_SLUK_LUTUTSKYLL  ; V8212  TIL SLUK I LUT-SKYLL ETTER AT  KONSENTRASJONEN HAR VAERT UNDER  GRENSEVERDI
LD TR0
AND V8212_HJ1
ANDNOT K2_TR20_TID_S  ; KURS 2 TRINN 20 TID
ANDNOT K2_NOEDSTOPP  ; VASKEPROGR. STOPPER OG PUMPENE I VASKEN STOPPER.
AND K2_TR06_TID_S  ; KURS 2 TRINN 06 TID
ANDNOT VST80_K2_V8212_SLUK_LUTUTSKYLL  ; V8212  TIL SLUK I LUT-SKYLL ETTER AT  KONSENTRASJONEN HAR VAERT UNDER  GRENSEVERDI
OUT V8212_HJ2
LD TR0
LD V8212_HJ2
LD V8212_FORS_INN  ; TID SOM FORSINKER  VENTIL AAPNING TIL T82 NAAR LUTKONSENTASJON ER OK FOERSTE GANG
AND K2_VASK_INNE
ANDNOT K2_TR21_TID_S  ; KURS 2 TRINN 21 TID
ORLD
ANDLD
TIM 0154 #50  ; TID SOM RESETSIGN. LIGGER INNE
LD TR0
AND V8212_HJ2
AND Q8017_RESETTID  ; TID SOM RESETSIGN. LIGGER INNE
LDNOT K2_VENT_TEMPERATUR
OR VST80_K2_SIRKULASJON_
ANDLD
OUT V8212_UT  ; Z

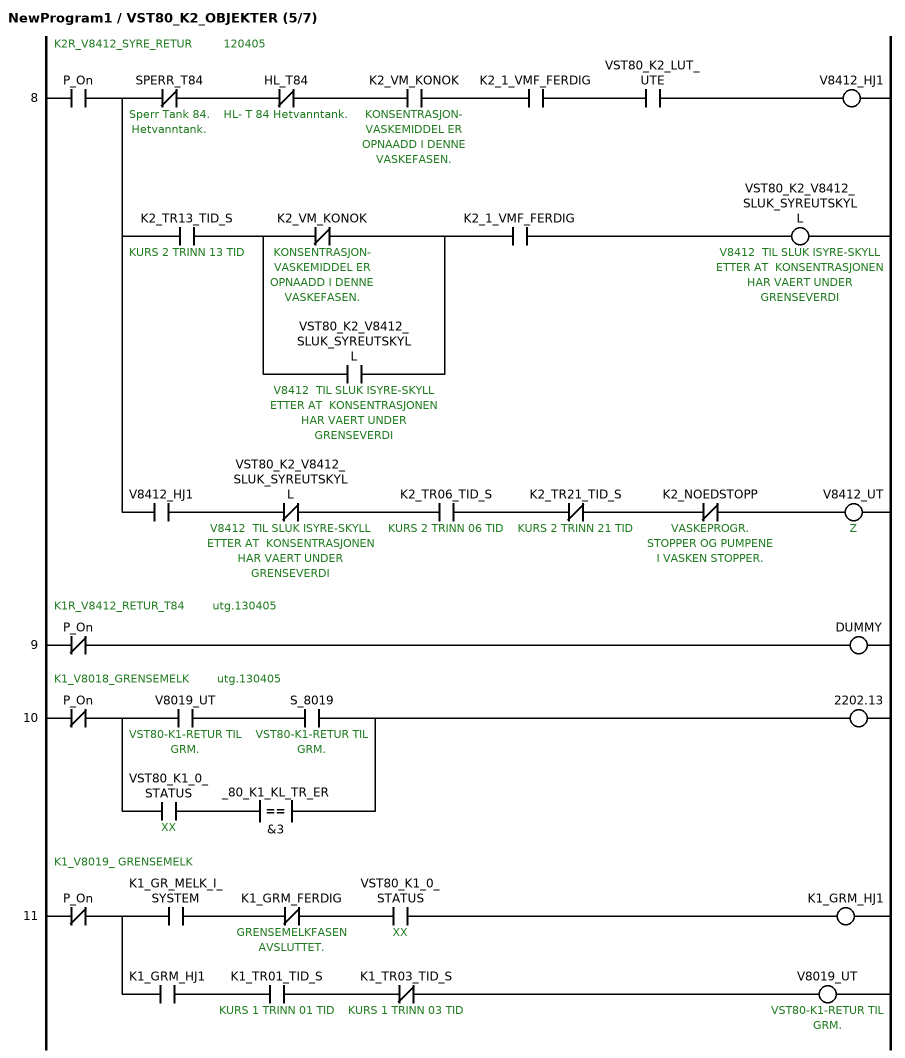
; rung 8: K2R_V8412_SYRE_RETUR         120405
LD P_On
OUT TR0
ANDNOT SPERR_T84  ; Sperr Tank 84. Hetvanntank.
ANDNOT HL_T84  ; HL- T 84 Hetvanntank.
AND K2_VM_KONOK  ; KONSENTRASJON-VASKEMIDDEL ER OPNAADD I DENNE VASKEFASEN.
AND K2_1_VMF_FERDIG
AND VST80_K2_LUT_UTE
OUT V8412_HJ1
LD TR0
AND K2_TR13_TID_S  ; KURS 2 TRINN 13 TID
LDNOT K2_VM_KONOK  ; KONSENTRASJON-VASKEMIDDEL ER OPNAADD I DENNE VASKEFASEN.
OR VST80_K2_V8412_SLUK_SYREUTSKYLL  ; V8412  TIL SLUK ISYRE-SKYLL ETTER AT  KONSENTRASJONEN HAR VAERT UNDER  GRENSEVERDI
ANDLD
AND K2_1_VMF_FERDIG
OUT VST80_K2_V8412_SLUK_SYREUTSKYLL  ; V8412  TIL SLUK ISYRE-SKYLL ETTER AT  KONSENTRASJONEN HAR VAERT UNDER  GRENSEVERDI
LD TR0
AND V8412_HJ1
ANDNOT VST80_K2_V8412_SLUK_SYREUTSKYLL  ; V8412  TIL SLUK ISYRE-SKYLL ETTER AT  KONSENTRASJONEN HAR VAERT UNDER  GRENSEVERDI
AND K2_TR06_TID_S  ; KURS 2 TRINN 06 TID
ANDNOT K2_TR21_TID_S  ; KURS 2 TRINN 21 TID
ANDNOT K2_NOEDSTOPP  ; VASKEPROGR. STOPPER OG PUMPENE I VASKEN STOPPER.
OUT V8412_UT  ; Z
; rung 9: K1R_V8412_RETUR_T84        utg.130405
LDNOT P_On
OUT DUMMY
; rung 10: K1_V8018_GRENSEMELK        utg.130405
LDNOT P_On
LD V8019_UT  ; VST80-K1-RETUR TIL GRM.
AND S_8019  ; VST80-K1-RETUR TIL GRM.
LD VST80_K1_0_STATUS  ; XX
AND=(300) _80_K1_KL_TR_ER &3
ORLD
ANDLD
OUT 2202.13
; rung 11: K1_V8019_GRENSEMELK
LDNOT P_On
OUT TR0
AND K1_GR_MELK_I_SYSTEM
ANDNOT K1_GRM_FERDIG  ; GRENSEMELKFASEN AVSLUTTET.
AND VST80_K1_0_STATUS  ; XX
OUT K1_GRM_HJ1
LD TR0
AND K1_GRM_HJ1
AND K1_TR01_TID_S  ; KURS 1 TRINN 01 TID
ANDNOT K1_TR03_TID_S  ; KURS 1 TRINN 03 TID
OUT V8019_UT  ; VST80-K1-RETUR TIL GRM.

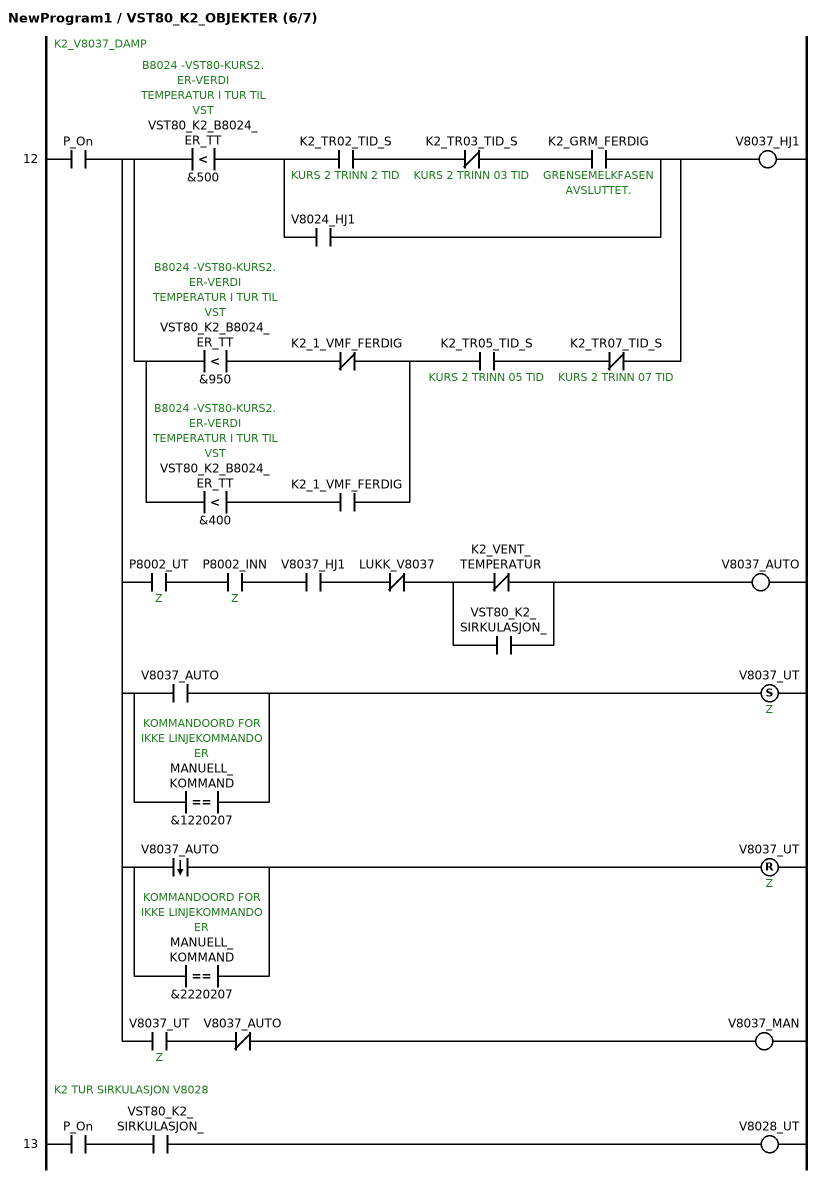
; rung 12: K2_V8037_DAMP
LD P_On
OUT TR0
LD<(310) VST80_K2_B8024_ER_TT &500  ; B8024 -VST80-KURS2. ER-VERDI TEMPERATUR I TUR TIL VST
LD K2_TR02_TID_S  ; KURS 2 TRINN 2 TID
ANDNOT K2_TR03_TID_S  ; KURS 2 TRINN 03 TID
AND K2_GRM_FERDIG  ; GRENSEMELKFASEN AVSLUTTET.
OR V8024_HJ1
ANDLD
LD<(310) VST80_K2_B8024_ER_TT &950  ; B8024 -VST80-KURS2. ER-VERDI TEMPERATUR I TUR TIL VST
ANDNOT K2_1_VMF_FERDIG
LD<(310) VST80_K2_B8024_ER_TT &400  ; B8024 -VST80-KURS2. ER-VERDI TEMPERATUR I TUR TIL VST
AND K2_1_VMF_FERDIG
ORLD
AND K2_TR05_TID_S  ; KURS 2 TRINN 05 TID
ANDNOT K2_TR07_TID_S  ; KURS 2 TRINN 07 TID
ORLD
ANDLD
OUT V8037_HJ1
LD TR0
AND P8002_UT  ; Z
AND P8002_INN  ; Z
AND V8037_HJ1
ANDNOT LUKK_V8037
LDNOT K2_VENT_TEMPERATUR
OR VST80_K2_SIRKULASJON_
ANDLD
OUT V8037_AUTO
LD TR0
LD V8037_AUTO
OR=L(301) MANUELL_KOMMAND &1220207  ; KOMMANDOORD FOR IKKE LINJEKOMMANDOER
ANDLD
SET V8037_UT  ; Z
LD TR0
%LD V8037_AUTO
OR=L(301) MANUELL_KOMMAND &2220207  ; KOMMANDOORD FOR IKKE LINJEKOMMANDOER
ANDLD
RSET V8037_UT  ; Z
LD TR0
AND V8037_UT  ; Z
ANDNOT V8037_AUTO
OUT V8037_MAN
; rung 13: K2 TUR SIRKULASJON V8028
LD P_On
AND VST80_K2_SIRKULASJON_
OUT V8028_UT

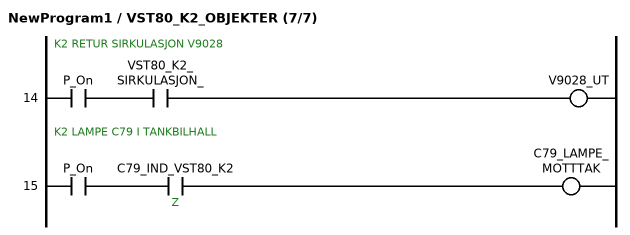
; rung 14: K2 RETUR SIRKULASJON V9028
LD P_On
AND VST80_K2_SIRKULASJON_
OUT V9028_UT
; rung 15: K2 LAMPE C79 I TANKBILHALL
LD P_On
AND C79_IND_VST80_K2  ; Z
OUT C79_LAMPE_MOTTTAK

### Section VST80_K2_KLAPRING
; VST80-KURS1 KLAPREPROGRAM

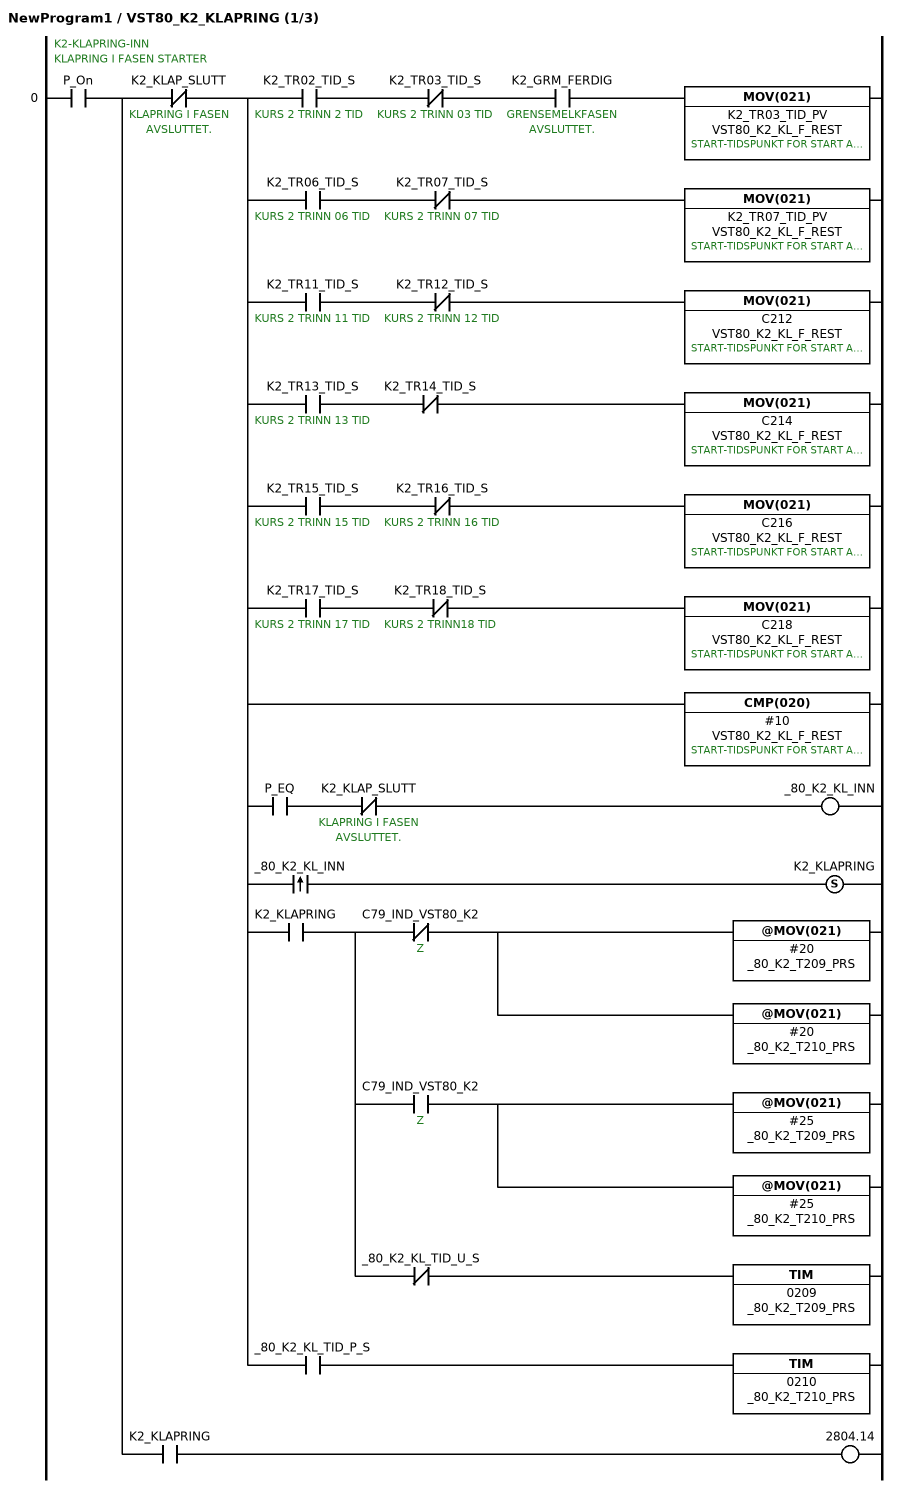
; rung 0: K2-KLAPRING-INN / KLAPRING I FASEN STARTER
LD P_On
OUT TR0
ANDNOT K2_KLAP_SLUTT  ; KLAPRING I FASEN AVSLUTTET.
OUT TR1
AND K2_TR02_TID_S  ; KURS 2 TRINN 2 TID
ANDNOT K2_TR03_TID_S  ; KURS 2 TRINN 03 TID
AND K2_GRM_FERDIG  ; GRENSEMELKFASEN AVSLUTTET.
MOV(021) K2_TR03_TID_PV VST80_K2_KL_F_REST  ; START-TIDSPUNKT FOR START AV KLAPRING
LD TR1
AND K2_TR06_TID_S  ; KURS 2 TRINN 06 TID
ANDNOT K2_TR07_TID_S  ; KURS 2 TRINN 07 TID
MOV(021) K2_TR07_TID_PV VST80_K2_KL_F_REST  ; START-TIDSPUNKT FOR START AV KLAPRING
LD TR1
AND K2_TR11_TID_S  ; KURS 2 TRINN 11 TID
ANDNOT K2_TR12_TID_S  ; KURS 2 TRINN 12 TID
MOV(021) C212 VST80_K2_KL_F_REST  ; START-TIDSPUNKT FOR START AV KLAPRING
LD TR1
AND K2_TR13_TID_S  ; KURS 2 TRINN 13 TID
ANDNOT K2_TR14_TID_S
MOV(021) C214 VST80_K2_KL_F_REST  ; START-TIDSPUNKT FOR START AV KLAPRING
LD TR1
AND K2_TR15_TID_S  ; KURS 2 TRINN 15 TID
ANDNOT K2_TR16_TID_S  ; KURS 2 TRINN 16 TID
MOV(021) C216 VST80_K2_KL_F_REST  ; START-TIDSPUNKT FOR START AV KLAPRING
LD TR1
AND K2_TR17_TID_S  ; KURS 2 TRINN 17 TID
ANDNOT K2_TR18_TID_S  ; KURS 2 TRINN18 TID
MOV(021) C218 VST80_K2_KL_F_REST  ; START-TIDSPUNKT FOR START AV KLAPRING
LD TR1
CMP(020) #10 VST80_K2_KL_F_REST  ; START-TIDSPUNKT FOR START AV KLAPRING
AND P_EQ
ANDNOT K2_KLAP_SLUTT  ; KLAPRING I FASEN AVSLUTTET.
OUT _80_K2_KL_INN
LD TR1
@AND _80_K2_KL_INN
SET K2_KLAPRING
LD TR1
AND K2_KLAPRING
OUT TR2
ANDNOT C79_IND_VST80_K2  ; Z
@MOV(021) #20 _80_K2_T209_PRS
@MOV(021) #20 _80_K2_T210_PRS
LD TR2
AND C79_IND_VST80_K2  ; Z
@MOV(021) #25 _80_K2_T209_PRS
@MOV(021) #25 _80_K2_T210_PRS
LD TR2
ANDNOT _80_K2_KL_TID_U_S
TIM 0209 _80_K2_T209_PRS
LD TR1
AND _80_K2_KL_TID_P_S
TIM 0210 _80_K2_T210_PRS
LD TR0
AND K2_KLAPRING
OUT 2804.14

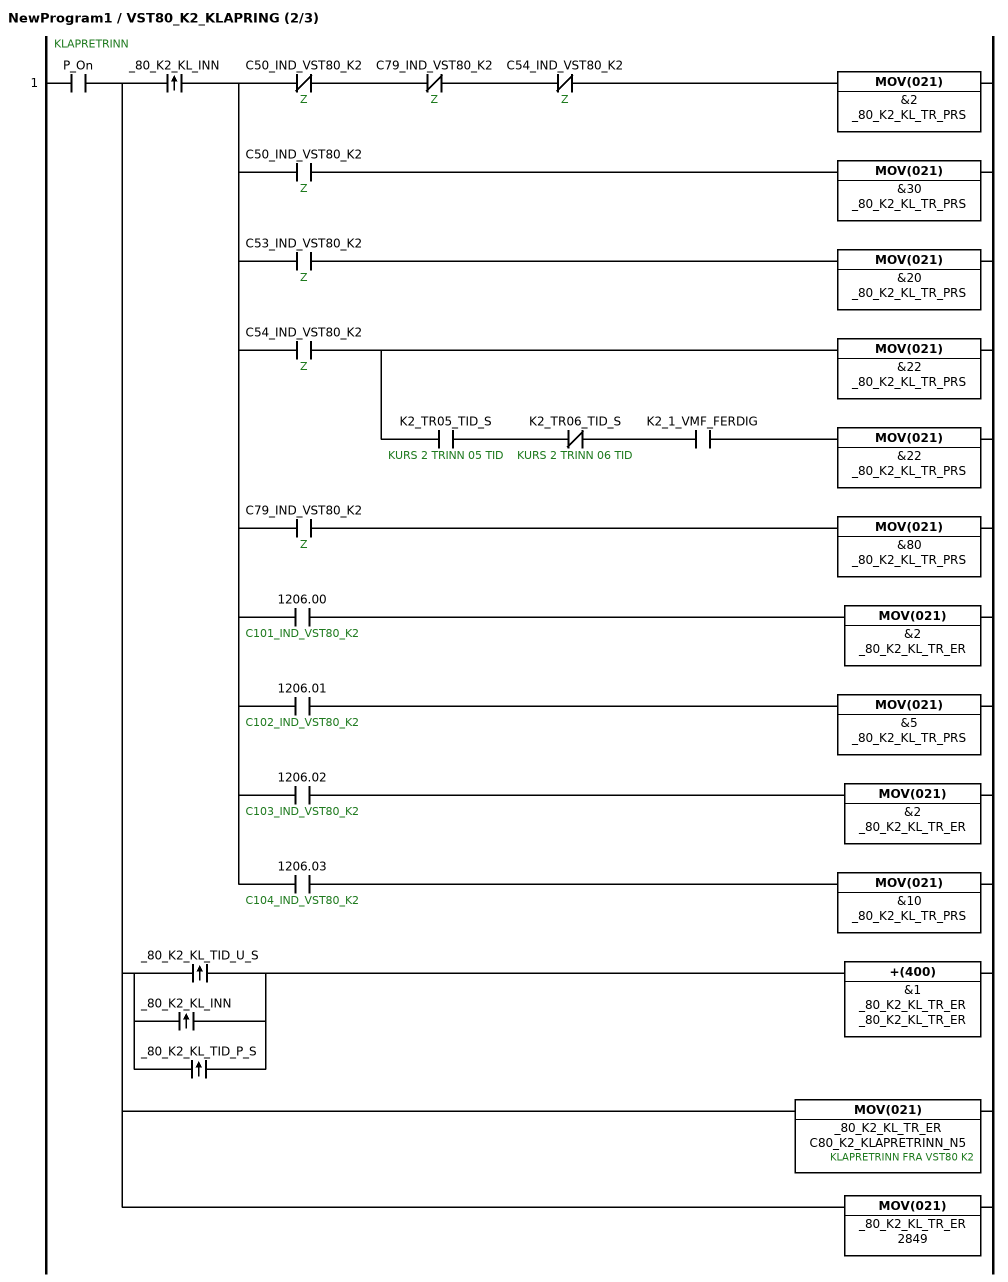
; rung 1: KLAPRETRINN
LD P_On
OUT TR0
@AND _80_K2_KL_INN
OUT TR1
ANDNOT C50_IND_VST80_K2  ; Z
ANDNOT C79_IND_VST80_K2  ; Z
ANDNOT C54_IND_VST80_K2  ; Z
MOV(021) &2 _80_K2_KL_TR_PRS
LD TR1
AND C50_IND_VST80_K2  ; Z
MOV(021) &30 _80_K2_KL_TR_PRS
LD TR1
AND C53_IND_VST80_K2  ; Z
MOV(021) &20 _80_K2_KL_TR_PRS
LD TR1
AND C54_IND_VST80_K2  ; Z
MOV(021) &22 _80_K2_KL_TR_PRS
AND K2_TR05_TID_S  ; KURS 2 TRINN 05 TID
ANDNOT K2_TR06_TID_S  ; KURS 2 TRINN 06 TID
AND K2_1_VMF_FERDIG
MOV(021) &22 _80_K2_KL_TR_PRS
LD TR1
AND C79_IND_VST80_K2  ; Z
MOV(021) &80 _80_K2_KL_TR_PRS
LD TR1
AND 1206.00  ; C101_IND_VST80_K2
MOV(021) &2 _80_K2_KL_TR_ER
LD TR1
AND 1206.01  ; C102_IND_VST80_K2
MOV(021) &5 _80_K2_KL_TR_PRS
LD TR1
AND 1206.02  ; C103_IND_VST80_K2
MOV(021) &2 _80_K2_KL_TR_ER
LD TR1
AND 1206.03  ; C104_IND_VST80_K2
MOV(021) &10 _80_K2_KL_TR_PRS
LD TR0
@LD _80_K2_KL_TID_U_S
@OR _80_K2_KL_INN
@OR _80_K2_KL_TID_P_S
ANDLD
+(400) &1 _80_K2_KL_TR_ER _80_K2_KL_TR_ER
LD TR0
MOV(021) _80_K2_KL_TR_ER C80_K2_KLAPRETRINN_N5  ; KLAPRETRINN FRA VST80 K2
MOV(021) _80_K2_KL_TR_ER 2849

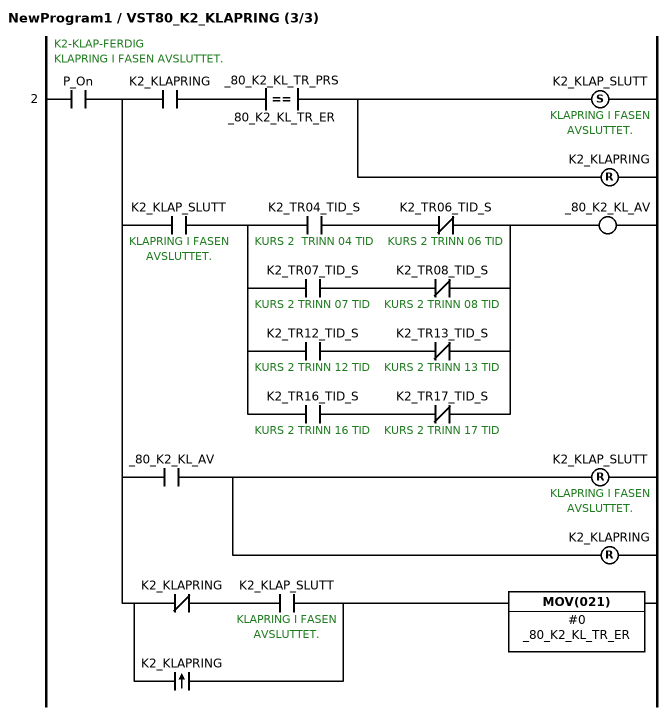
; rung 2: K2-KLAP-FERDIG / KLAPRING I FASEN AVSLUTTET.
LD P_On
OUT TR0
AND K2_KLAPRING
AND=(300) _80_K2_KL_TR_PRS _80_K2_KL_TR_ER
SET K2_KLAP_SLUTT  ; KLAPRING I FASEN AVSLUTTET.
RSET K2_KLAPRING
LD TR0
AND K2_KLAP_SLUTT  ; KLAPRING I FASEN AVSLUTTET.
LD K2_TR04_TID_S  ; KURS 2  TRINN 04 TID
ANDNOT K2_TR06_TID_S  ; KURS 2 TRINN 06 TID
LD K2_TR07_TID_S  ; KURS 2 TRINN 07 TID
ANDNOT K2_TR08_TID_S  ; KURS 2 TRINN 08 TID
ORLD
LD K2_TR12_TID_S  ; KURS 2 TRINN 12 TID
ANDNOT K2_TR13_TID_S  ; KURS 2 TRINN 13 TID
ORLD
LD K2_TR16_TID_S  ; KURS 2 TRINN 16 TID
ANDNOT K2_TR17_TID_S  ; KURS 2 TRINN 17 TID
ORLD
ANDLD
OUT _80_K2_KL_AV
LD TR0
AND _80_K2_KL_AV
RSET K2_KLAP_SLUTT  ; KLAPRING I FASEN AVSLUTTET.
RSET K2_KLAPRING
LD TR0
LDNOT K2_KLAPRING
AND K2_KLAP_SLUTT  ; KLAPRING I FASEN AVSLUTTET.
@OR K2_KLAPRING
ANDLD
MOV(021) #0 _80_K2_KL_TR_ER

### Section VST80_K2_GRAF_TR_
; OVERFØRING AV TRINN I VASK TIL GRAFIKK

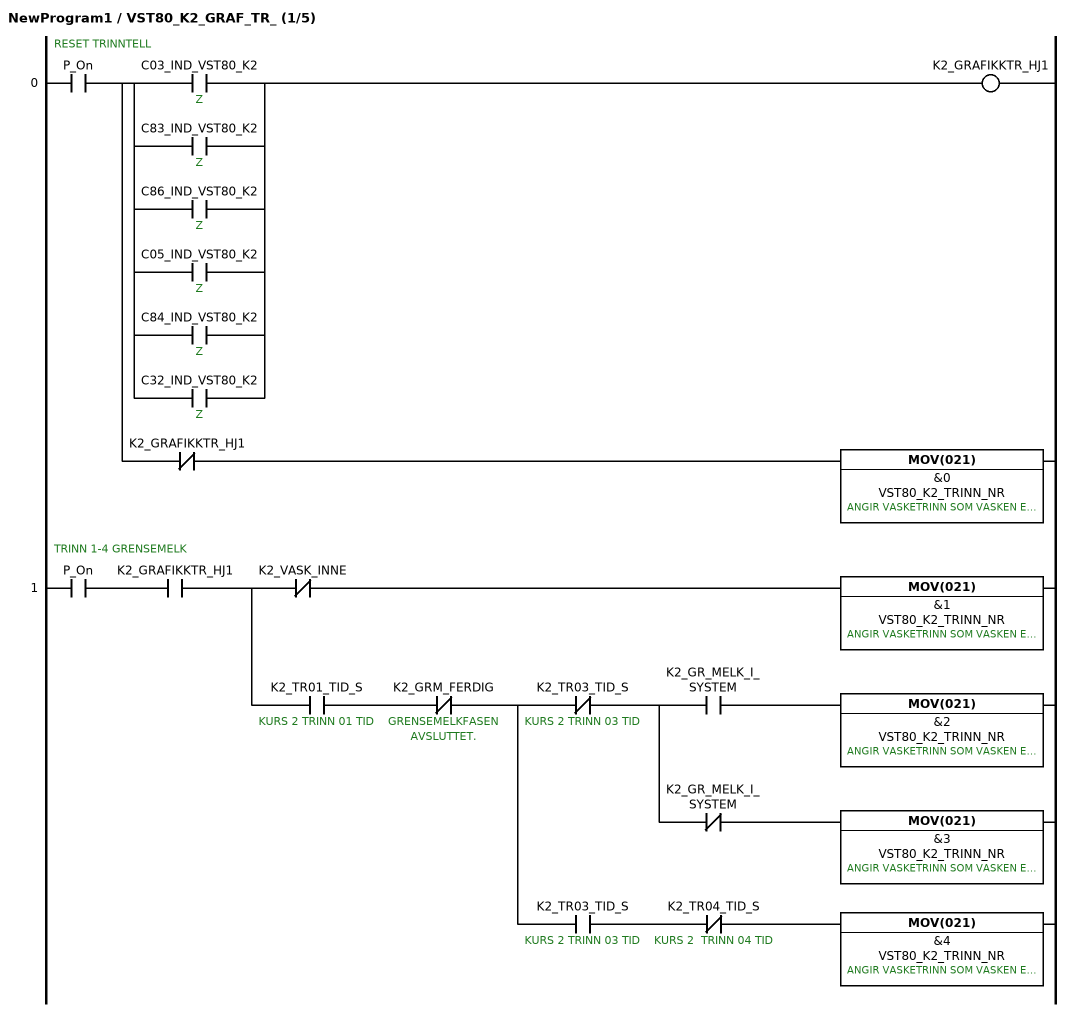
; rung 0: RESET TRINNTELL
LD P_On
OUT TR0
LD C03_IND_VST80_K2  ; Z
OR C83_IND_VST80_K2  ; Z
OR C86_IND_VST80_K2  ; Z
OR C05_IND_VST80_K2  ; Z
OR C84_IND_VST80_K2  ; Z
OR C32_IND_VST80_K2  ; Z
ANDLD
OUT K2_GRAFIKKTR_HJ1
LD TR0
ANDNOT K2_GRAFIKKTR_HJ1
MOV(021) &0 VST80_K2_TRINN_NR  ; ANGIR VASKETRINN SOM VASKEN ER I
; rung 1: TRINN 1-4 GRENSEMELK
LD P_On
AND K2_GRAFIKKTR_HJ1
OUT TR0
ANDNOT K2_VASK_INNE
MOV(021) &1 VST80_K2_TRINN_NR  ; ANGIR VASKETRINN SOM VASKEN ER I
LD TR0
AND K2_TR01_TID_S  ; KURS 2 TRINN 01 TID
ANDNOT K2_GRM_FERDIG  ; GRENSEMELKFASEN AVSLUTTET.
OUT TR0
ANDNOT K2_TR03_TID_S  ; KURS 2 TRINN 03 TID
OUT TR1
AND K2_GR_MELK_I_SYSTEM
MOV(021) &2 VST80_K2_TRINN_NR  ; ANGIR VASKETRINN SOM VASKEN ER I
LD TR1
ANDNOT K2_GR_MELK_I_SYSTEM
MOV(021) &3 VST80_K2_TRINN_NR  ; ANGIR VASKETRINN SOM VASKEN ER I
LD TR0
AND K2_TR03_TID_S  ; KURS 2 TRINN 03 TID
ANDNOT K2_TR04_TID_S  ; KURS 2  TRINN 04 TID
MOV(021) &4 VST80_K2_TRINN_NR  ; ANGIR VASKETRINN SOM VASKEN ER I

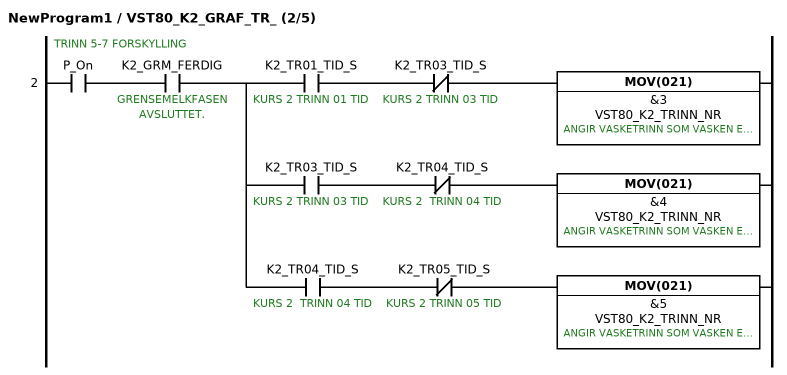
; rung 2: TRINN 5-7 FORSKYLLING
LD P_On
AND K2_GRM_FERDIG  ; GRENSEMELKFASEN AVSLUTTET.
OUT TR0
AND K2_TR01_TID_S  ; KURS 2 TRINN 01 TID
ANDNOT K2_TR03_TID_S  ; KURS 2 TRINN 03 TID
MOV(021) &3 VST80_K2_TRINN_NR  ; ANGIR VASKETRINN SOM VASKEN ER I
LD TR0
AND K2_TR03_TID_S  ; KURS 2 TRINN 03 TID
ANDNOT K2_TR04_TID_S  ; KURS 2  TRINN 04 TID
MOV(021) &4 VST80_K2_TRINN_NR  ; ANGIR VASKETRINN SOM VASKEN ER I
LD TR0
AND K2_TR04_TID_S  ; KURS 2  TRINN 04 TID
ANDNOT K2_TR05_TID_S  ; KURS 2 TRINN 05 TID
MOV(021) &5 VST80_K2_TRINN_NR  ; ANGIR VASKETRINN SOM VASKEN ER I

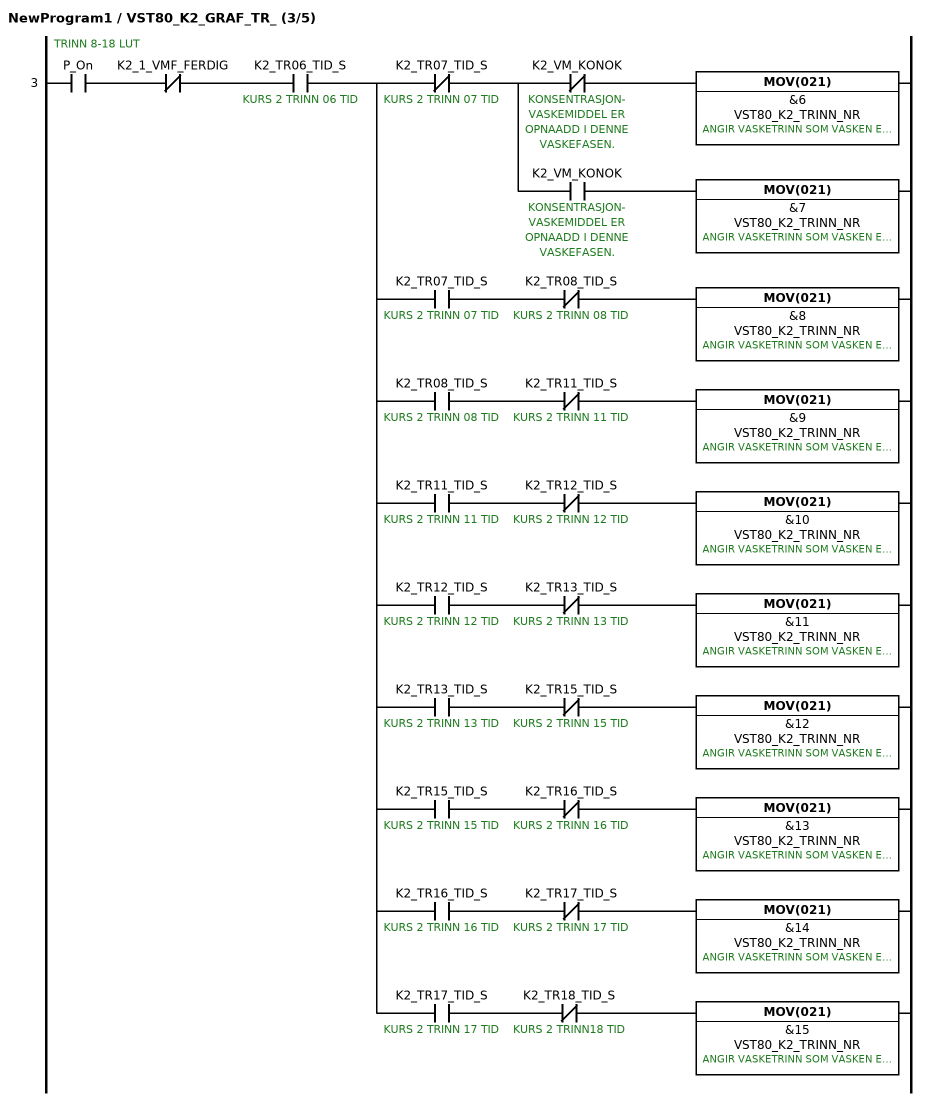
; rung 3: TRINN 8-18 LUT
LD P_On
ANDNOT K2_1_VMF_FERDIG
AND K2_TR06_TID_S  ; KURS 2 TRINN 06 TID
OUT TR0
ANDNOT K2_TR07_TID_S  ; KURS 2 TRINN 07 TID
OUT TR1
ANDNOT K2_VM_KONOK  ; KONSENTRASJON-VASKEMIDDEL ER OPNAADD I DENNE VASKEFASEN.
MOV(021) &6 VST80_K2_TRINN_NR  ; ANGIR VASKETRINN SOM VASKEN ER I
LD TR1
AND K2_VM_KONOK  ; KONSENTRASJON-VASKEMIDDEL ER OPNAADD I DENNE VASKEFASEN.
MOV(021) &7 VST80_K2_TRINN_NR  ; ANGIR VASKETRINN SOM VASKEN ER I
LD TR0
AND K2_TR07_TID_S  ; KURS 2 TRINN 07 TID
ANDNOT K2_TR08_TID_S  ; KURS 2 TRINN 08 TID
MOV(021) &8 VST80_K2_TRINN_NR  ; ANGIR VASKETRINN SOM VASKEN ER I
LD TR0
AND K2_TR08_TID_S  ; KURS 2 TRINN 08 TID
ANDNOT K2_TR11_TID_S  ; KURS 2 TRINN 11 TID
MOV(021) &9 VST80_K2_TRINN_NR  ; ANGIR VASKETRINN SOM VASKEN ER I
LD TR0
AND K2_TR11_TID_S  ; KURS 2 TRINN 11 TID
ANDNOT K2_TR12_TID_S  ; KURS 2 TRINN 12 TID
MOV(021) &10 VST80_K2_TRINN_NR  ; ANGIR VASKETRINN SOM VASKEN ER I
LD TR0
AND K2_TR12_TID_S  ; KURS 2 TRINN 12 TID
ANDNOT K2_TR13_TID_S  ; KURS 2 TRINN 13 TID
MOV(021) &11 VST80_K2_TRINN_NR  ; ANGIR VASKETRINN SOM VASKEN ER I
LD TR0
AND K2_TR13_TID_S  ; KURS 2 TRINN 13 TID
ANDNOT K2_TR15_TID_S  ; KURS 2 TRINN 15 TID
MOV(021) &12 VST80_K2_TRINN_NR  ; ANGIR VASKETRINN SOM VASKEN ER I
LD TR0
AND K2_TR15_TID_S  ; KURS 2 TRINN 15 TID
ANDNOT K2_TR16_TID_S  ; KURS 2 TRINN 16 TID
MOV(021) &13 VST80_K2_TRINN_NR  ; ANGIR VASKETRINN SOM VASKEN ER I
LD TR0
AND K2_TR16_TID_S  ; KURS 2 TRINN 16 TID
ANDNOT K2_TR17_TID_S  ; KURS 2 TRINN 17 TID
MOV(021) &14 VST80_K2_TRINN_NR  ; ANGIR VASKETRINN SOM VASKEN ER I
LD TR0
AND K2_TR17_TID_S  ; KURS 2 TRINN 17 TID
ANDNOT K2_TR18_TID_S  ; KURS 2 TRINN18 TID
MOV(021) &15 VST80_K2_TRINN_NR  ; ANGIR VASKETRINN SOM VASKEN ER I

